// TIA Portal project "Program_PLC_LEGO" (V18)

(* hardware
DEVICE "S7-1200 station_1"  S7-1200 Station
   slot 0: "Rack_0"  S7-1200 Rack  Rack  V1.0
   slot 1: "PLC_1"  CPU 1214C DC/DC/DC  6ES7 214-1AG40-0XB0  V4.6
DEVICE "master"  GSD.Device.PN
   slot 0: "Rack"  Rack  V1.0
   slot 0: "bnixg35080b5r067"  BNI XG3-508-0B5-R067  BNI00L3  V1.3.2
      slot 0: "BNI XG3-508-0B5-R067"  BNI XG3-508-0B5-R067
      slot 1: "PN-IO"  PN-IO
         slot 1: "Port XF1"  Port XF1
         slot 2: "Port XF2"  Port XF2
   slot 1: "IO-Link I/O Ports_1"  IO-Link I/O Ports
      slot 0: "BALLUFF 8 Port IO-Link Master"  BALLUFF 8 Port IO-Link Master
   slot 1: "Digital Input"  Digital Input
   slot 2: "Digital Input_1"  Digital Input
   slot 3: "IOL_I/O_10/10_Byte + PQI_2"  IOL_I/O_10/10_Byte + PQI
   slot 4: "IOL_I/O_10/10_Byte + PQI_3"  IOL_I/O_10/10_Byte + PQI
   slot 5: "IOL_I/O_10/10_Byte + PQI_1"  IOL_I/O_10/10_Byte + PQI
   slot 6: "IOL_I/O_10/10_Byte + PQI"  IOL_I/O_10/10_Byte + PQI
   slot 7: "BNI IOL-302-S02-X026"  BNI IOL-302-S02-X026
   slot 8: "IOL_I/O_32/32_Byte + PQI"  IOL_I/O_32/32_Byte + PQI
*)

// ===== PLC "PLC_1"  CPU 1214C DC/DC/DC =====

VAR_GLOBAL   // PLC tag table "Default tag table"
   "Tag_1" AT %I68.0 : Bool;
   "Tag_2" AT %I68.1 : Bool;
   "RFID1" AT %I96.0 : Bool;   // rfid1
   "Tag_4" AT %M10.0 : Bool;
   "Tag_5" AT %ID98 : DWord;
   "Tag_6" AT %QB96 : Byte;
   "Tag_7" AT %M10.1 : Bool;
   "RFID2" AT %I107.0 : Bool;
   "RFID3" AT %I85.0 : Bool;
   "RFID4" AT %I74.0 : Bool;
   "Tag_8" AT %I68.2 : Bool;
   "Tag_9" AT %I68.3 : Bool;
   "Tag_10" AT %I3.0 : Bool;
   "Tag_11" AT %I4.0 : Bool;
END_VAR

TYPE "udtZlecenia"
   STRUCT
      Zlecenie : Struct
         ID : Int;   // Numer zlecenia
         Model : Int;   // Rodzaj modelu 2-8
         PartNo : Int;   // Nr sztuki
         "Time" : Struct   // Czasy na stanowiskach
            Stanowisko1 : Struct
               StartTime : DTL;   // Czas rozpoczecia
               EndTime : DTL;   // Czas zakonczenia
               TargetTime : Int;   // Zakladany czas
               ActualTime : Int;
               Abort : Bool;   // Czy anulowano produkcje na tym stanowisku
            END_STRUCT;
            Stanowisko2 : Struct
               StartTime : DTL;   // Czas rozpoczecia
               EndTime : DTL;   // Czas zakonczenia
               TargetTime : Int;   // Zakladany czas
               ActualTime : Int;
               Abort : Bool;   // Czy anulowano produkcje na tym stanowisku
            END_STRUCT;
            Stanowisko3 : Struct
               StartTime : DTL;   // Czas rozpoczecia
               EndTime : DTL;   // Czas zakonczenia
               TargetTime : Int;   // Zakladany czas
               ActualTime : Int;
               Abort : Bool;   // Czy anulowano produkcje na tym stanowisku
            END_STRUCT;
            StanowiskoQC : Struct
               StartTime : DTL;   // Czas rozpoczecia
               EndTime : DTL;   // Czas zakonczenia
               TargetTime : Int;   // Zakladany czas
               ActualTime : Int;
               Abort : Bool;   // Czy anulowano produkcje na tym stanowisku
            END_STRUCT;
         END_STRUCT;
         Alarm : Struct
            Stanowisko1 : Struct
               MissingPart : Bool;
               DamagedPart : Bool;
               PalletFault : Bool;
               WrongInstruction : Bool;
               SensorFault : Bool;
               Other : Bool;
            END_STRUCT;
            Stanowisko2 : Struct
               MissingPart : Bool;
               DamagedPart : Bool;
               PalletFault : Bool;
               WrongInstruction : Bool;
               SensorFault : Bool;
               Other : Bool;
            END_STRUCT;
            Stanowisko3 : Struct
               MissingPart : Bool;
               DamagedPart : Bool;
               PalletFault : Bool;
               WrongInstruction : Bool;
               SensorFault : Bool;
               Other : Bool;
            END_STRUCT;
            StanowieskoQC : Struct
               Camera : Bool;
               NOK : Bool;
               PalletFault : Bool;
               RFID : Bool;
               SensorFault : Bool;
               Other : Bool;
            END_STRUCT;
         END_STRUCT;
         ReturnQC : Bool;   // True - poprawny wyrób, False zły wyrób
         Priority : Int;   // 0 - Najniższy, 5 - Najwyższy
         Status : Array[0..3] of Bool;   // Status czy skonczono na danym stanowisku
         NOK : Struct
            NoBrick : Bool;
            WrongColour : Bool;
            Offset : Bool;
            Damage : Bool;
            WrongNumber : Bool;
            Other : Bool;
         END_STRUCT;
      END_STRUCT;
   END_STRUCT;
END_TYPE

TYPE "udtStanowiskoAssembly"
   STRUCT
      Config : Struct
         ID : Int;
         "Name" : String[20];
         HorlyRate : Real;
      END_STRUCT;
      Production : Struct
         State : Int;   // 0 - Gotowy. 1 - Montaż, 2 - Zakończono, 3 - Awaria
         OrderNo : Int;
         ProductNo : Int;
      END_STRUCT;
      "Time" : Struct
         TargetTime : Time;
         LastSec : UInt;
         RemainingSec : Int;
         RemainingStr : String[6];
         Blink : Bool;
      END_STRUCT;
      Commands : Struct
         Start : Struct
            Enable : Bool;
            State : Bool;
         END_STRUCT;
         FInish : Struct
            Enable : Bool;
            State : Bool;
         END_STRUCT;
         ReportFault : Struct
            Enable : Bool;
            State : Bool;
         END_STRUCT;
         AbortProcess : Struct
            Enable : Bool;
            State : Bool;
         END_STRUCT;
         FaultReason : Struct
            MissingPart : Bool;
            DamagedPart : Bool;
            PalletFault : Bool;
            WrongInstruction : Bool;
            SensorFault : Bool;
            Other : Bool;
         END_STRUCT;
      END_STRUCT;
      Sensors : Struct
         PalletPresent : Bool;
         RFID : Struct
            TagPresent : Bool;
            CmdRead : Bool;
            CmdWrite : Bool;
            Status : Bool;
            OrderNo : Int;
            ProductNo : Int;
         END_STRUCT;
      END_STRUCT;
      Stats : Struct
         DoneToday : Int;
         Efficiency : Int;
         ActudalPart : Int;
         Instruction : Int;
         Loaded : Bool;
      END_STRUCT;
      HMI : Struct
         Clear : Bool;   // Czyści licznik
         Container : Array[1..3] of Struct   // Tablica kontenerów
            value : Int;   // Ilość kontenerów 0 - 3
            Add : Struct   // Impuls na reczne dodanie
               Enable : Bool;
               Status : Bool;
            END_STRUCT;
            Subtract : Struct   // Impuls na reczne odejmowanie
               Enable : Bool;
               Status : Bool;
            END_STRUCT;
         END_STRUCT;
      END_STRUCT;
      MontazState : Int;
   END_STRUCT;
END_TYPE

TYPE "udtDbKomunikacja"
   STRUCT
      Trigger : Bool;
      NumerZlecenia : String[50];
      NumerOperacji : DInt;
      NumerPaletki : String[50];
      Stanowisko : String[50];
      Operator : String[50];
      CzasCykluMs : DInt;
      WynikQC : Bool;
      IloscWyprodukowanych : DInt;
      LiczbaWadliwych : DInt;
      KodPostoju : String[20];
   END_STRUCT;
END_TYPE

DATA_BLOCK "DB_Data"   // DB1
{ S7_Optimized_Access := 'FALSE' }
VERSION : 0.1
   VAR
      Stanowisko1 : "udtStanowiskoAssembly";
      Stanowisko2 : "udtStanowiskoAssembly";
      Stanowisko3 : "udtStanowiskoAssembly";
      StanowiskoQC : Struct
         Config : Struct
            ID : Int;
            "Name" : String[20];
            HorlyRate : Real;
         END_STRUCT;
         Production : Struct
            State : Int;
            OrderNo : Int;
            ProductNo : Int;
         END_STRUCT;
         "Time" : Struct
            TargetTime : Time;
            LastSec : UInt;
            RemainingSec : Int;
            RemainingStr : String[6];
            Blink : Bool;
         END_STRUCT;
         Commands : Struct
            Start : Struct
               Enable : Bool;
               State : Bool;
            END_STRUCT;
            OK : Struct
               Enable : Bool;
               State : Bool;
            END_STRUCT;
            NOK : Struct
               Enable : Bool;
               State : Bool;
               NoBrick : Bool;
               WrongColour : Bool;
               Offset : Bool;
               Damage : Bool;
               WrongNumber : Bool;
               Other : Bool;
            END_STRUCT;
            ReportFault : Struct
               Enable : Bool;
               State : Bool;
            END_STRUCT;
         END_STRUCT;
         Sensors : Struct
            PalletPresent : Bool;
            RFID : Struct
               TagPresent : Bool;
               CmdRead : Bool;
               CmdWrite : Bool;
               Status : Bool;
               OrderNo : Int;
               ProductNo : Int;
            END_STRUCT;
         END_STRUCT;
         Stats : Struct
            DoneToday : Int;
            Efficiency : Int;
            ActudalPart : Int;
            Instruction : Int;
            Loaded : Bool;
            PartsOK : Int;
            PartsNOK : Int;
            PartsPercent : Int;
         END_STRUCT;
         HMI : Struct
            Clear : Bool;
            CameraStatus : Int;
         END_STRUCT;
         QualityState : Int;
         FaultReason : Struct
            Camera : Bool;
            NOK : Bool;
            PalletFault : Bool;
            RFID : Bool;
            SensorFault : Bool;
            Other : Bool;
         END_STRUCT;
         CameraControl : Struct
            bInit : Bool;
            bGetResult : Bool;
            bResetError : Bool;
            wynikOK : Bool;
            bReq : Bool;
            bTrigger : Bool;
            bZrobInspekcje : Bool;
            krok : Int;
            wynikOV : Array[0..5] of Bool;
            CameraStatus : Bool;
         END_STRUCT;
      END_STRUCT;
      ZlecenieIndex : Array[0..3] of Int;
      DoneAllTime : Array[0..3] of Int;
   END_VAR
BEGIN
   Stanowisko1.Production.State := 0;
   Stanowisko1.Production.OrderNo := 0;   // Nr zlecenia
   // Stanowisko1.Config.ID : ID stanowiska
   // Stanowisko1.Config."Name" : Nazwa stanowiska
   // Stanowisko1.Config.HorlyRate : Stawka godzinowa
   // Stanowisko1.Production.ProductNo : Nr modelu
   // Stanowisko1."Time".TargetTime : Zakładany czas ukończenia wyrobu
   // Stanowisko1."Time".RemainingSec : pozostałe sekundy
   // Stanowisko1."Time".RemainingStr : sekundy w string
   // Stanowisko1.Commands : komendy
END_DATA_BLOCK

DATA_BLOCK "DB_PTL"   // DB2
{ S7_Optimized_Access := 'FALSE' }
VERSION : 0.1
   VAR
      PTL_state : Array[0..8] of Bool;
      Stanowisko : Array[0..2] of Struct
         Row1 : Int;   // 0 - brak, 3 - wszytskie kontenery
         Row2 : Int;   // 0 - brak, 3 - wszytskie kontenery
         Row3 : Int;   // 0 - brak, 3 - wszytskie kontenery
      END_STRUCT;
      ConnParams : TCON_IP_v4;
      InitDone : Bool;
      Wyzwalacz : Bool;
      mb_done : Bool;
      mb_busy : Bool;
      mb_error : Bool;
      mb_status : Word;
      PTL_Buttons : Array[1..9] of Word;
      PTL_State_Old : Array[0..8] of Bool;
   END_VAR
BEGIN
   // PTL_state[0] : Stanowisko 1.1
   // PTL_state[1] : Stanowisko 1.2
   // PTL_state[2] : Stanowisko 1.3
   // PTL_state[3] : Stanowisko 2.1
   // PTL_state[4] : Stanowisko 2.2
   // PTL_state[5] : Stanowisko 2.3
   // PTL_state[6] : Stanowisko 3.1
   // PTL_state[7] : Stanowisko 3.2
   // PTL_state[8] : Stanowisko 3.3
END_DATA_BLOCK

DATA_BLOCK "DB_Zlecenia"   // DB3
{ S7_Optimized_Access := 'FALSE' }
VERSION : 0.1
   VAR
      Zlecenie : Array[0..199] of "udtZlecenia";
      NastepneZlecenie : "udtZlecenia";
      PusteZlecenie : "udtZlecenia";   // Nie dopisywac wartosci!!!
      ResetZlecen : Bool;
   END_VAR
BEGIN
END_DATA_BLOCK

DATA_BLOCK "DB_WWW"   // DB5
{ S7_Optimized_Access := 'FALSE' }
VERSION : 0.1
   VAR
      Comm : "udtDbKomunikacja";
   END_VAR
BEGIN
END_DATA_BLOCK

DATA_BLOCK "BIS_V_CLM_COM_DB"   // DB6
{ S7_Optimized_Access := 'TRUE' }
AUTHOR : BICU
FAMILY : Ident
VERSION : 1.0
// stored: InstanceOfName BIS_V_CLM_COM
"BIS_V_CLM_COM"
BEGIN
END_DATA_BLOCK

DATA_BLOCK "RFID_test"   // DB7
{ S7_Optimized_Access := 'TRUE' }
VERSION : 0.1
   VAR
      Bufor_Odczyt : Array[0..10] of Byte;
      Bufor_Zapis : Array[0..10] of Byte;
      Bufor_Odczyt2 : Array[0..10] of Byte;
      Bufor_Odczyt3 : Array[0..10] of Byte;
      Bufor_Odczyt4 : Array[0..10] of Byte;
   END_VAR
BEGIN
END_DATA_BLOCK

DATA_BLOCK "BIS_V_CLM_COM_DB_1"   // DB8
{ S7_Optimized_Access := 'TRUE' }
AUTHOR : BICU
FAMILY : Ident
VERSION : 1.0
// stored: InstanceOfName BIS_V_CLM_COM
"BIS_V_CLM_COM"
BEGIN
END_DATA_BLOCK

DATA_BLOCK "BIS_V_CLM_COM_DB_2"   // DB9
{ S7_Optimized_Access := 'TRUE' }
AUTHOR : BICU
FAMILY : Ident
VERSION : 1.0
// stored: InstanceOfName BIS_V_CLM_COM
"BIS_V_CLM_COM"
BEGIN
END_DATA_BLOCK

DATA_BLOCK "DB_Cam_Input"   // DB10
{ S7_Optimized_Access := 'FALSE' }
VERSION : 0.1
   VAR
      Input : Array[0..127] of Byte;
   END_VAR
BEGIN
END_DATA_BLOCK

DATA_BLOCK "DB_Cam_Output"   // DB11
{ S7_Optimized_Access := 'FALSE' }
VERSION : 0.1
   VAR
      Output : Array[0..127] of Byte;
   END_VAR
BEGIN
END_DATA_BLOCK

DATA_BLOCK "BVS_Sensor_DB"   // DB12
{ S7_Optimized_Access := 'TRUE' }
AUTHOR : PD-ILS
FAMILY : Balluff
VERSION : 1.1
// stored: InstanceOfName BVS_Sensor
"BVS_Sensor"
BEGIN
END_DATA_BLOCK

DATA_BLOCK "BIS_V_CLM_COM_DB_3"   // DB13
{ S7_Optimized_Access := 'TRUE' }
AUTHOR : BICU
FAMILY : Ident
VERSION : 1.0
// stored: InstanceOfName BIS_V_CLM_COM
"BIS_V_CLM_COM"
BEGIN
END_DATA_BLOCK

FUNCTION_BLOCK "RaportowanieDB"   // FB1, SCL
{ S7_Optimized_Access := 'TRUE' }
VERSION : 0.1
   VAR_TEMP
      temp_CzasObecny : Int;
      temp_DTL : Int;
      temp_RoznicaCzasu : Time;
   END_VAR
BEGIN
   // Uruchamiaj tylko, gdy C# potwierdził odebranie poprzednich danych (Trigger = 0)
   IF NOT "DB_WWW".Comm.Trigger THEN

       // ============================================
       // STANOWISKO 1 (Montażowe)
       // ============================================
       IF "DB_Data".Stanowisko1.Commands.FInish.State THEN

          // #temp_CzasObecny := RD_SYS_T(OUT => #temp_DTL);
          // #temp_RoznicaCzasu := T_DIFF(IN1 := #temp_DTL, IN2 := "DB_Data".Stanowisko1."Time".StartStamp);
           "DB_WWW".Comm.CzasCykluMs := TIME_TO_DINT(#temp_RoznicaCzasu);

           "DB_WWW".Comm.NumerZlecenia := 'ZL-2137'; // do podmiany na aktualne zlecenie
           "DB_WWW".Comm.Stanowisko := 'Assembly 1';
           "DB_WWW".Comm.Operator := 'Operator 1';
           "DB_WWW".Comm.IloscWyprodukowanych := 1;

           IF "DB_Data".Stanowisko1.Commands.FaultReason.DamagedPart THEN
               "DB_WWW".Comm.KodPostoju := 'DAMAGED_PART';
               "DB_WWW".Comm.WynikQC := FALSE;
               "DB_WWW".Comm.LiczbaWadliwych := 1;
           ELSIF "DB_Data".Stanowisko1.Commands.FaultReason.MissingPart THEN
               "DB_WWW".Comm.KodPostoju := 'MISSING_PART';
               "DB_WWW".Comm.WynikQC := FALSE;
               "DB_WWW".Comm.LiczbaWadliwych := 1;
           ELSE
               "DB_WWW".Comm.KodPostoju := '';
               "DB_WWW".Comm.WynikQC := TRUE;
               "DB_WWW".Comm.LiczbaWadliwych := 0;
           END_IF;

           "DB_WWW".Comm.Trigger := TRUE;
           "DB_Data".Stanowisko1.Production.State := 2;
           "DB_Data".Stanowisko1.Commands.FInish.State := FALSE;

           // ============================================
           // STANOWISKO 2 (Montażowe)
           // ============================================
         //  ELSIF "DB_Data".Stanowisko2.Commands.FInish.State THEN

           //    #temp_CzasObecny := RD_SYS_T(OUT => #temp_DTL);
           //    #temp_RoznicaCzasu := T_DIFF(IN1 := #temp_DTL, IN2 := "DB_Data".Stanowisko2."Time".StartStamp);
            //   "DB_WWW".Comm.CzasCykluMs := TIME_TO_DINT(#temp_RoznicaCzasu);

            //   "DB_WWW".Comm.NumerZlecenia := 'ZL-2137';
            //   "DB_WWW".Comm.Stanowisko := 'Assembly 2';
            //   "DB_WWW".Comm.Operator := 'Operator 2';
            //   "DB_WWW".Comm.IloscWyprodukowanych := 1;

            //   IF "DB_Data".Stanowisko2.Commands.FaultReason.DamagedPart THEN
            //       "DB_WWW".Comm.KodPostoju := 'DAMAGED_PART';
            //       "DB_WWW".Comm.WynikQC := FALSE;
             //      "DB_WWW".Comm.LiczbaWadliwych := 1;
            //   ELSIF "DB_Data".Stanowisko2.Commands.FaultReason.MissingPart THEN
           //        "DB_WWW".Comm.KodPostoju := 'MISSING_PART';
           //        "DB_WWW".Comm.WynikQC := FALSE;
           //        "DB_WWW".Comm.LiczbaWadliwych := 1;
           //    ELSE
           //        "DB_WWW".Comm.KodPostoju := '';
           //        "DB_WWW".Comm.WynikQC := TRUE;
           //        "DB_WWW".Comm.LiczbaWadliwych := 0;
            //   END_IF;

            //   "DB_WWW".Comm.Trigger := TRUE;
            //   "DB_Data".Stanowisko2.Production.State := 2;
            //   "DB_Data".Stanowisko2.Commands.FInish.State := FALSE;

               // ============================================
               // STANOWISKO 3 (Montażowe)
               // ============================================
         //  ELSIF "DB_Data".Stanowisko3.Commands.FInish.State THEN

            //   #temp_CzasObecny := RD_SYS_T(OUT => #temp_DTL);
            //   #temp_RoznicaCzasu := T_DIFF(IN1 := #temp_DTL, IN2 := "DB_Data".Stanowisko3."Time".StartStamp);
            //   "DB_WWW".Comm.CzasCykluMs := TIME_TO_DINT(#temp_RoznicaCzasu);

            //   "DB_WWW".Comm.NumerZlecenia := 'ZL-2137';
           //    "DB_WWW".Comm.Stanowisko := 'Assembly 3';
            //   "DB_WWW".Comm.Operator := 'Operator 3';
            //   "DB_WWW".Comm.IloscWyprodukowanych := 1;

           //    IF "DB_Data".Stanowisko3.Commands.FaultReason.DamagedPart THEN
           //        "DB_WWW".Comm.KodPostoju := 'DAMAGED_PART';
            //       "DB_WWW".Comm.WynikQC := FALSE;
             //      "DB_WWW".Comm.LiczbaWadliwych := 1;
            //   ELSIF "DB_Data".Stanowisko3.Commands.FaultReason.MissingPart THEN
            //       "DB_WWW".Comm.KodPostoju := 'MISSING_PART';
           //        "DB_WWW".Comm.WynikQC := FALSE;
           ///        "DB_WWW".Comm.LiczbaWadliwych := 1;
           //    ELSE
           //        "DB_WWW".Comm.KodPostoju := '';
           //        "DB_WWW".Comm.WynikQC := TRUE;
           //        "DB_WWW".Comm.LiczbaWadliwych := 0;
           //    END_IF;

           //    "DB_WWW".Comm.Trigger := TRUE;
            //   "DB_Data".Stanowisko3.Production.State := 2;
             //  "DB_Data".Stanowisko3.Commands.FInish.State := FALSE;

               // ============================================
               // STANOWISKO 4 (QC - Kontrola Jakości)
               // ============================================
         //  ELSIF "DB_Data".StanowiskoQC.Commands.FInish.State THEN

             //  #temp_CzasObecny := RD_SYS_T(OUT => #temp_DTL);
             //  #temp_RoznicaCzasu := T_DIFF(IN1 := #temp_DTL, IN2 := "DB_Data".StanowiskoQC."Time".StartStamp);
            //   "DB_WWW".Comm.CzasCykluMs := TIME_TO_DINT(#temp_RoznicaCzasu);

             //  "DB_WWW".Comm.NumerZlecenia := 'ZL-2137';
             //  "DB_WWW".Comm.Stanowisko := 'QC Station';
             //  "DB_WWW".Comm.Operator := 'Operator QC';

               // Zależnie od tego, jak raportujecie odrzuty na QC
              // IF "DB_Data".StanowiskoQC.Commands.FaultReason.DamagedPart THEN
              //     "DB_WWW".Comm.IloscWyprodukowanych := 0;
              //     "DB_WWW".Comm.KodPostoju := 'DAMAGED_PART';
              //     "DB_WWW".Comm.WynikQC := FALSE;
              //     "DB_WWW".Comm.LiczbaWadliwych := 1;
              // ELSE
              //     "DB_WWW".Comm.IloscWyprodukowanych := 1;
               //    "DB_WWW".Comm.KodPostoju := '';
               //    "DB_WWW".Comm.WynikQC := TRUE;
             //      "DB_WWW".Comm.LiczbaWadliwych := 0;
             //  END_IF;

             //  "DB_WWW".Comm.Trigger := TRUE;
               //"DB_Data".StanowiskoQC.Production.State := 2;
               //"DB_Data".StanowiskoQC.Commands.FInish.State := FALSE;

       END_IF;

   END_IF;
END_FUNCTION_BLOCK

FUNCTION_BLOCK "BIS_V_CLM_COM"   // FB33, SCL
TITLE = BIS V (VM, C, VL), BIS C, BIS M; BIS L Function Block
{ S7_Optimized_Access := 'TRUE' }
AUTHOR : BICU
FAMILY : Ident
VERSION : 1.0
   VAR_INPUT
      Init : Bool := FALSE;   // Internal reset and initailisation of FB
      Start : Bool := FALSE;   // Start command
      ProcReset : Bool := FALSE;   // Reset of BIS and FB
      HeadOff : Bool := FALSE;   // Head deactivation
      Dynamic : Bool := FALSE;   // Dynamic read / write function
      HW_LADDR : Hw_SubModule;   // HW_Address for cyclic com, BIS Module
      HW_LADDR_Q : Hw_SubModule;   // HW_Address for cyclic com, BIS Output Module
      Command : Int := 0;   // 1=Read; 2=Write;
      DB_Send : DB_ANY;
      Offset_DBSend : DInt := 0;   // Offset write data
      DB_Receive : DB_ANY;
      Offset_DBReceive : DInt := 0;   // Offset read data
      TAG_StartAddr : DInt := DINT#0;   // Start address from data carrier or parameter number
      TAG_NumbOfByte : DInt := DINT#0;   // Data lenght to be written or read or parameter Bytes
      WatchdogTime : Time := T#3S;   // Watchdog of commado
      CopTargetAddr : DInt;   // Traget Address for Copy Command
      CopRW_HeadNo : Int;   // Head number for Copy Command
      ProcType : Char := 'v';   // Processor Type V= BIS-V only | C, L, M = BIS * | I = BIS-M4** IO-Link
      OptIoLen : UInt := 10;   // Optional IO Length for IO-Link and C, L, M
      OptIoBuffOffs : UInt;   // IO Buffer offset for BIS C, L, M, 2nd R/W head
   END_VAR
   VAR_OUTPUT
      Ready : Bool := FALSE;   // Command ready
      Error : Bool := FALSE;   // Command error
      ErrorCode : Word := 0;   // Error code
      MT : Bool := FALSE;   // Antenna selection is on
      DatCarrPresent : Bool := FALSE;   // Data Carrier present
   END_VAR
   VAR_IN_OUT
      DB_SendOpt : Variant;   // Data block write data
      DB_ReceiveOpt : Variant;   // Data block for read data
   END_VAR
   VAR
      PointerByte : DInt := 0;   // Pointer DB RW-Address
      LengthByte : DInt := 0;   // Number of bytes read/write per cycle
      BytePerPage : DInt := 0;   // Databytes lenght in IO buffer
      TotalByte : DInt := 0;   // Remaining all Byte data to be read/write
      HW_Init : Bool;   // Hardware adresses initialized
      ReadActive : Bool := FALSE;   // Read command active
      WriteActive : Bool := FALSE;   // Write command active
      ResetActive : Bool := FALSE;   // FB and Processor reset active
      ToggleOld : Bool := FALSE;   // Last state toggle-bit
      FirstCycle : Bool := FALSE;   // First read/write cycle
      IMP_Start : Bool := FALSE;   // Pulse bit Start
      ShortCom : Bool := FALSE;   // Command with 1 Byte data-length active
      RdLengIn : Bool;   // Read length info from input
      WriteCom : Bool := FALSE;   // Write command without data active
      CopyTag : Bool := FALSE;   // Copy Tag commando
      HeadOffActive : Bool := FALSE;   // AntSelBusy
      WaitOnAE : Bool;   // Read on AE Bit
      IOLink_Proc : Bool;   // BIS IO-Link processor M-4**-0**-001
      IOLink_Proc401 : Bool;   // BIS IO-Link processor M-4**-0**-401
      CLM_Proc : Bool;   // BIS classic C, L, M processor unit
      C_Cttp : Bool;   // BIS C Tag Type. False 32 Byte. True 64 Byte
      bHd_CP_CodePresent : Bool;   // Bit header In: Tag Present
      bHd_AA_JobStart : Bool;   // Bit header In: Job Start
      bHd_AE_JobEnd : Bool;   // Bit header In: Job End
      bHd_AF_JobError : Bool;   // Bit header In: Job Error
      bHd_MT_MultTag : Bool;   // Bit header In: Multiple Tags
      bHd_TO_ToggleOut : Bool;   // Bit header In: Toggle Bit Out
      bHd_HF_HeadFault : Bool;   // Bit header In: Head Fault
      bHd_BB_Ready : Bool;   // Bit header In: Ready for Operation
      bHd_AV_JobStart : Bool;   // Bit header Out: Job Start
      bHd_GR_Default : Bool;   // Bit header Out: Default State
      bHd_HD_HeadSel : Bool;   // Bit header Out: Head Selection BIS U
      bHd_KA_HeadOff : Bool;   // Bit header Out: Head shutoff
      bHd_TI_ToggleIn : Bool;   // Bit header Out: Togle Bit In
      bHd_Cttp_TagType : Bool;
      ProcRes_Int : Bool;   // Processor reset internal
      ErrorInt : Bool;   // Error bit internal
      ArrayInput : Array[0..#InBuSi] of Byte;   // BIS out to PLC in
      ArrayOutput : Array[0..#OutBuSi] of Byte;   // PLC out to BIS in
      R_TRIG_Start : R_TRIG;
      R_TRIG_Reset : R_TRIG;
      R_TRIG_KA : R_TRIG;
      F_TRIG_KA : F_TRIG;
      WD_Timer : TON_TIME;
      HF_Timer : TON_TIME;
      PIaddr : UDInt;   // Input address
      PIcount : UInt;   // Input length
      PQaddr : UDInt;   // Output address
      PQcount : UInt;   // Output address
      RetVal_ModulDiag : Int;   // Return value modul diagnosis
      RetVal_RD_Addr : Int;   // Return value read address
      RetVal_RD_DP : Int;   // Return value read input data
      RetVal_WR_DP : Int;   // Return value write output data
      RetVal_Get_ErrID : Word;   // Return value get error ID
      RetValVarMove : Int;
      CNT_Diag : UInt;   // CNT_Modul Diag
      Diag_Out : DWord;   // Modul Diag
      BIS_STA : Struct   // BIS Statusword
         CP_DaCarrPres : Bool := FALSE;   // Data Carrier present
         reserved_1 : Bool := FALSE;
         reserved_2 : Bool := FALSE;
         reserved_3 : Bool := FALSE;
         ChainedCom : Bool := FALSE;
         reserved_5 : Bool := FALSE;
         Error : Bool := FALSE;   // Error output set
         Ready : Bool := FALSE;   // FB Ready
         ResetAct : Bool := FALSE;   // Reset running
         Command_start : Bool := FALSE;   // FB Start is set
         reserved_6 : Bool := FALSE;
         InitAct : Bool := TRUE;   // Init running
         HF_Bit : Bool := FALSE;   // Head fault
         Busy : Bool := FALSE;   // Comando busy
         Reserved_7 : Bool := FALSE;
         Reserved_8 : Bool := FALSE;
         Com : Int := 0;   // 81=Read;82=Write; 42=Read EPC; 44=Read TID
         TStartAddr : DInt := DINT#0;   // Start address from data carrier or parameter number for diagnosis
         TNumbOfByte : DInt := DINT#0;   // data lenght to be written or read or parameter Bytes for diagnosis
      END_STRUCT;
      testdword : DWord;
   END_VAR
   VAR_TEMP
      tError : Word;   // temp Error number buffer
      tBTimeoutIN : Bool;   // temp Timeout in
      tBTimeoutQ : Bool;   // temp Timeout output
      tLoop : DInt;   // temp Loop counter
      tempDB : DB_ANY;
      tUdint : UDInt;
      tLCnt : UDInt;
      tVariant : Variant;
      tErrorConvVar : Int;
      tempTest : DB_ANY;
      tWordTest : Word;
      tempDBErr : Int;
   END_VAR
   VAR CONSTANT
      InBuSi : Int := 254;   // maximum size inputbuffer
      OutBuSi : Int := 254;   // maximum size outputbuffer
   END_VAR
BEGIN
   //=============================================================================
   //Balluff GmbH
   //(c)Copyright (2019) All Rights Reserved
   //-----------------------------------------------------------------------------
   //Library: BIS_V
   //Tested with: CPU 1214C V4.1
   //Engineering: TIA Portal V13 SP1 
   //Restrictions: -
   //Requirements: PLC (S7-1200 / S7-1500)
   //Functionality: RFID commandos for BIS V, BIS C, BIS M, BIS L processor units
   //-----------------------------------------------------------------------------
   //Change log table:
   //Version  Date       Expert in charge  Changes applied
   //
   //00.01.00 18.03.2019 Balluff GmbH PD   First created with TIA V13 SP1 with mem opt
   //=============================================================================
   //
   (*
   Disclaimer of Liability
   **********************
   The demo function block is free of charge and is a universal application 
   example.
   This demo function block shall help program and configure PLC applications and 
   shall provide possible solutions.
   The user is not entitled to claim for warranty, error correction and updates. 
   In 
   particular there is excluded any claims against Balluff GmbH for damages that 
   might result from the use of this demo program. Excluded from this limitation 
   of 
   liability shall be (a) those damages that are based on injury to life, limb or 
   health, (b) a liability according to the Produkthaftungsgesetz (German Product 
   Liability Law) and (c) cases of willful intent.
   Please check if the function block is intended for your application before 
   adapting it in plants and machineries.
   By using the S7 sample, made available free of charge you accept the limitation 
   of 
   warranty and liability!

   Haftungsausschluss:
   *********************
   Der hier kostenlos verfügbare DEMO-Baustein ist ein allgemeingültiges 
   Anwendungsbeispiel. Dieser DEMO-Baustein soll bei der Programmierung und 
   Projektierung von SPS-Anwendungen unterstützen und Lösungsansätze aufzeigen. 
   Ein Anspruch auf Gewährleistung, Fehlerbeseitigung und Update besteht für den 
   Anwender nicht. Die BALLUFF GmbH schließt insbesondere jegliche Haftung für 
   Schäden, die durch den Einsatz dieses DEMO-Bausteins entstehen, ausdrücklich 
   aus! Diese Haftungsbeschränkung gilt nicht bei Verletzungen des Lebens, des 
   Körpers oder der Gesundheit, bei der Haftung nach dem Produkthaftungsgesetz und 
   bei vorsätzlichen Pflichtverletzungen. 
   Prüfen Sie vor dem Einsatz in Anlagen und Maschinen, ob der hier 
   bereitgestellte 
   DEMO Baustein für Ihre Anwendung nutzbar ist!
   Mit dem Einsatz des hier kostenlos vorgelegten S7-Beispiel erkennen Sie die 
   Gewährleistungs- und Haftungsbegrenzung an!

       *)

   //-----------------------------------------------------------------------------
   //Select Processor unit
   //-----------------------------------------------------------------------------


   // Default select BIS V
   IF (#ProcType = 'V') OR
     (#ProcType = 'v') THEN
     #WaitOnAE := FALSE;
     #IOLink_Proc := FALSE;
     #CLM_Proc := FALSE;
     #IOLink_Proc401 := FALSE;

     // Select BIS C, L, M processor    
   ELSIF (#ProcType = 'M') OR // M upper case
     (#ProcType = 'm') OR // m lower case
     (#ProcType = 'C') OR // C upper case
     (#ProcType = 'c') OR // c lower case
     (#ProcType = 'L') OR // L upper case
     (#ProcType = 'l') THEN // l lower case
     #WaitOnAE := TRUE;
     #IOLink_Proc := FALSE;
     #CLM_Proc := TRUE;
     #IOLink_Proc401 := FALSE;

     // Select BIS IO-Link compact processor unit    
   ELSIF (#ProcType = 'I') OR  // I upper case
     (#ProcType = 'i') THEN  // i lower case
     #WaitOnAE := TRUE;
     #IOLink_Proc := TRUE;
     #CLM_Proc := FALSE;
     #IOLink_Proc401 := FALSE;

     // Select BIS IO-Link compact processor unit   BIS M-4xx-xxx-401 
   ELSIF (#ProcType = 'K') OR  // I upper case
     (#ProcType = 'k') THEN  // i lower case
     #WaitOnAE := TRUE;
     #IOLink_Proc := TRUE;
     #CLM_Proc := FALSE;
     #IOLink_Proc401 := TRUE;

     // Siemens Master BIS M-4xx-xxx-001        
   ELSIF (#ProcType = 'X') OR  // I upper case
     (#ProcType = 'x') THEN  // i lower case
     #WaitOnAE := TRUE;
     #IOLink_Proc := TRUE;
     #CLM_Proc := TRUE;
     #IOLink_Proc401 := FALSE;

     // Siemens Master BIS M-4xx-xxx-401     
   ELSIF (#ProcType = 'Y') OR  // I upper case
     (#ProcType = 'y') THEN  // i lower case
     #WaitOnAE := TRUE;
     #IOLink_Proc := TRUE;
     #CLM_Proc := TRUE;
     #IOLink_Proc401 := TRUE;

   END_IF;

   // Select tag type for C System
   IF ((#ProcType = 'C') OR // C upper case
     (#ProcType = 'c')) AND // c lower case
     #C_Cttp THEN
     #bHd_Cttp_TagType := TRUE;
   ELSE
     #bHd_Cttp_TagType := FALSE;
   END_IF;

   //-------------------------------------------------
   // HMI Out
   //-------------------------------------------------
   #BIS_STA.CP_DaCarrPres := #bHd_CP_CodePresent;
   #BIS_STA.HF_Bit := #bHd_HF_HeadFault;
   #BIS_STA.InitAct := #Init;
   #BIS_STA.Error := #ErrorInt;

   #BIS_STA.ResetAct := #ResetActive;
   //-----------------------------------------------------------------------------
   //FB Init, reset static variables
   //-----------------------------------------------------------------------------
   IF #Init THEN
     #PointerByte := 0;
     #LengthByte := 0;
     #BytePerPage := 0;
     #TotalByte := 0;
     #ReadActive := FALSE;
     #WriteActive := FALSE;
     #ResetActive := FALSE;
     #ToggleOld := FALSE;
     #FirstCycle := FALSE;
     #ShortCom := FALSE;
     #WriteCom := FALSE;
     #Ready := TRUE;
     #Error := FALSE;
     #ErrorCode := 0;
     #HW_Init := FALSE;
     #HeadOffActive := FALSE;
     #ProcRes_Int := TRUE;
     #R_TRIG_Reset.Stat_Bit := FALSE;
   END_IF;

   //-----------------------------------------------------------------------------
   // read modul states
   //-----------------------------------------------------------------------------
   #RetVal_ModulDiag := GET_DIAG(MODE := 0, LADDR := #HW_LADDR, CNT_DIAG => #CNT_Diag, DIAG := #Diag_Out);

   //-----------------------------------------------------------------------------
   // reading PI/PQ addr and data length
   //-----------------------------------------------------------------------------
   IF NOT #HW_Init THEN
     #RetVal_RD_Addr := RD_ADDR(LADDR := #HW_LADDR, PIADDR => #PIaddr, PICount => #PIcount,
                                PQADDR => #PQaddr, PQCount => #PQcount);
     IF #IOLink_Proc THEN
       #PIcount := #OptIoLen;
       #PQcount := #OptIoLen;
     END_IF;

     IF #CLM_Proc THEN
       IF NOT #IOLink_Proc THEN
         #RetVal_RD_Addr := RD_ADDR(LADDR := #HW_LADDR_Q, PIADDR => #tUdint, PICount => #tUdint,
                                    PQADDR => #PQaddr, PQCount => #PQcount);
       END_IF;

       IF #OptIoBuffOffs = 0 THEN //1st Buffer selected
         #PQcount := #OptIoLen; // overwrite length
         #PIcount := #OptIoLen;
       ELSIF #OptIoBuffOffs <> 0 THEN //2nd Buffer selected
         #PQaddr := #PQaddr + #OptIoBuffOffs; // overwrite Address 
         #PQcount := #OptIoLen; // overwrite Address 
         #PIaddr := #PIaddr + #OptIoBuffOffs;
         #PIcount := #OptIoLen;
       END_IF;
     END_IF;

     #HW_Init := TRUE;
   END_IF;

   //-----------------------------------------------------------------------------
   // cyclic read cam input if HW init done
   //----------------------------------------------------------------------------- 
   IF #HW_Init THEN
     IF #CLM_Proc THEN
       #tLCnt := 0;
       #RetVal_RD_DP := 0;
       #RetVal_WR_DP := 0;
       FOR #tLoop := UDINT_TO_DINT(#PIaddr) TO UDINT_TO_DINT(#PIaddr + #PIcount) DO
         #ArrayInput[#tLCnt] := PEEK(area := 16#81, dbNumber := 0, byteOffset := #tLoop);
         #tLCnt := #tLCnt + 1;
       END_FOR;

     ELSE
       #RetVal_RD_DP := DPRD_DAT(LADDR := #HW_LADDR, RECORD => #ArrayInput);
     END_IF;
   END_IF;
   //-----------------------------------------------------------------------------
   // Comapre bitheader
   //-----------------------------------------------------------------------------
   IF #ArrayInput[0] <> #ArrayInput[#PIcount - 1] THEN
     RETURN;
   END_IF;

   //-----------------------------------------------------------------------------
   // Move input bytes to static bits
   //-----------------------------------------------------------------------------
   #bHd_CP_CodePresent := #ArrayInput[0].%X0;
   #bHd_AA_JobStart := #ArrayInput[0].%X1;
   #bHd_AE_JobEnd := #ArrayInput[0].%X2;
   #bHd_AF_JobError := #ArrayInput[0].%X3;
   #bHd_MT_MultTag := #ArrayInput[0].%X4;
   #bHd_TO_ToggleOut := #ArrayInput[0].%X5;
   #bHd_HF_HeadFault := #ArrayInput[0].%X6;
   #bHd_BB_Ready := #ArrayInput[0].%X7;

   //-------------------------------------------------
   // KA HeadOff
   //-------------------------------------------------
   #R_TRIG_KA(CLK := #HeadOff);
   #F_TRIG_KA(CLK := #HeadOff);
   IF #R_TRIG_KA.Q THEN    // Deactivate head
     #bHd_KA_HeadOff := TRUE;
     #Ready := FALSE;
     #DatCarrPresent := FALSE;
     #HeadOffActive := TRUE;
     GOTO DataOut;
   END_IF;

   IF #F_TRIG_KA.Q THEN    // Activate head
     #bHd_KA_HeadOff := FALSE;
     #Ready := FALSE;
     #HeadOffActive := FALSE;
     GOTO DataOut;
   END_IF;

   //-------------------------------------------------
   // FB Reset
   //-------------------------------------------------
   #R_TRIG_Reset(CLK := #ProcReset OR #ProcRes_Int);

   IF #R_TRIG_Reset.Q THEN
     #ResetActive := TRUE;
     #PointerByte := 0;
     #LengthByte := 0;
     #BytePerPage := 0;
     #TotalByte := 0;
     #ReadActive := FALSE;
     #WriteActive := FALSE;
     #ToggleOld := FALSE;
     #FirstCycle := FALSE;
     #ShortCom := FALSE;
     #WriteCom := FALSE;
     #CopyTag := FALSE;
     #Ready := FALSE;
     #bHd_GR_Default := TRUE;
     IF NOT #ProcRes_Int THEN
       #Error := FALSE;
       #ErrorCode := 0;
     END_IF;
     #ProcRes_Int := FALSE;
     #HeadOffActive := FALSE;
     GOTO DataOut;

   END_IF;

   IF #ResetActive AND NOT #bHd_BB_Ready THEN
     #bHd_GR_Default := false;
     #ResetActive := false;
     GOTO AV_Reset;
   END_IF;
   //-----------------------------------------------------------------------------
   // MT Multiple Tags; CT Present
   //-----------------------------------------------------------------------------
   #MT := #bHd_MT_MultTag;

   #DatCarrPresent := #bHd_CP_CodePresent;

   //-----------------------------------------------------------------------------
   // Command Start
   #R_TRIG_Start(CLK := #Start,
                 Q => #IMP_Start);
   //-----------------------------------------------------------------------------

   //-----------------------------------------------------------------------------
   // Check HW/Profinet Error when start is set
   //-----------------------------------------------------------------------------
   IF #IMP_Start THEN
     IF #RetVal_RD_Addr <> 0 THEN
       #tError := w#16#50; //Error read address
       GOTO Error;
     END_IF;

     IF #RetVal_RD_DP <> 0 THEN
       #tError := w#16#51; //Error read input data
       GOTO Error;
     END_IF;

     IF #RetVal_WR_DP <> 0 THEN
       #tError := w#16#52; //Error read output data
       GOTO Error;
     END_IF;

   END_IF;

   IF #bHd_AF_JobError AND NOT #ProcReset THEN // Check error
     #tError := #ArrayInput[1];
     GOTO Error;
   END_IF;

   #HF_Timer(IN := #bHd_HF_HeadFault AND (NOT #HeadOff OR (NOT #IOLink_Proc AND NOT #CLM_Proc)),
             PT := t#500ms);

   IF #HF_Timer.Q//Head fault timeout
     AND NOT #ProcReset
     AND (NOT #IOLink_Proc
     OR #IOLink_Proc
     AND NOT #HeadOff)
   THEN // Check head fault
     #tError := 16#09;
     GOTO Error;
   END_IF;

   IF #IMP_Start AND
     (#TAG_NumbOfByte > 65534) AND NOT
     (#Command = 16#B2) THEN
     #tError := w#16#84;
     GOTO Error;
   END_IF;

   //-----------------------------------------------------------------------------
   // FB ready output 
   //-----------------------------------------------------------------------------
   #Ready :=
   NOT #ReadActive AND
   NOT #WriteActive AND
   NOT #ResetActive AND
   NOT #ShortCom AND
   NOT #CopyTag AND
   NOT #WriteCom AND
   NOT #bHd_AA_JobStart AND
   NOT #bHd_AE_JobEnd AND
   NOT #bHd_AF_JobError AND
   NOT #HeadOffActive AND
   #bHd_BB_Ready;

   //-----------------------------------------------------------------------------
   // BIS status for HMI
   //-----------------------------------------------------------------------------
   #BIS_STA.Ready := #Ready;
   #BIS_STA.Command_start := #Start;
   #BIS_STA.Com := #Command;
   #BIS_STA.TStartAddr := #TAG_StartAddr;
   #BIS_STA.TNumbOfByte := #TAG_NumbOfByte;

   IF #BIS_STA.Ready THEN
     #BIS_STA.ResetAct := FALSE;
     #BIS_STA.Busy := FALSE;
   END_IF;
   //-----------------------------------------------------------------------------
   // Generate error timeout
   //-----------------------------------------------------------------------------
   #tBTimeoutIN := (NOT #Ready AND NOT #Dynamic
   AND NOT #ResetActive
   AND NOT #HeadOffActive
   AND NOT #ProcRes_Int);

   #WD_Timer(IN := #tBTimeoutIN,
             PT := #WatchdogTime,
             Q => #tBTimeoutQ);

   IF #tBTimeoutQ THEN
     #tError := w#16#80;
     #ProcRes_Int := #bHd_AA_JobStart;
     GOTO Error;
   END_IF;

   //=============================================================================
   //
   // Reader commandos
   //
   //=============================================================================

   //-----------------------------------------------------------------------------
   // Goto FB end if no job active
   //-----------------------------------------------------------------------------

   IF (NOT #ReadActive AND
     NOT #WriteActive AND
     NOT #ShortCom AND
     NOT #WriteCom AND
     NOT #CopyTag AND
     (NOT #IMP_Start OR
     NOT #Ready OR
     #bHd_AA_JobStart)) OR
     #HeadOffActive THEN
     RETURN;
   END_IF;

   IF #ReadActive THEN  // Check Get or Set
     GOTO Read;
   ELSIF #WriteActive THEN
     GOTO Write;
   ELSIF #WriteCom OR #CopyTag THEN
     GOTO WriteCom;
   END_IF;

   //-----------------------------------------------------------------------------
   // Initialize Command output
   //-----------------------------------------------------------------------------
   #ArrayOutput[3] := 0;
   #ArrayOutput[4] := 0;
   #ArrayOutput[5] := 0;
   #ArrayOutput[6] := 0;
   #ArrayOutput[7] := 0;
   #ArrayOutput[8] := 0;

   CASE #Command OF

     16#1: // Read user data       
       #ArrayOutput[1] := 16#1;
       #PointerByte := #Offset_DBReceive;
       #ReadActive := TRUE;
     16#2: // Write user data       
       #ArrayOutput[1] := 16#2;
       #PointerByte := #Offset_DBSend;
       #WriteActive := TRUE;
     16#7: // // Store Start address for Auto read
       #ArrayOutput[1] := 16#7;
       #WriteActive := TRUE;
       #WriteCom := TRUE;
     16#9: // Read Typ and Serial  
       #ArrayOutput[1] := 16#9;
       #PointerByte := #Offset_DBReceive;
       #RdLengIn := TRUE;
       #ReadActive := TRUE;
     16#11: // Copy data between data carriers
       #ArrayOutput[1] := 16#11;
       #PointerByte := #Offset_DBReceive;
       #WriteCom := TRUE;
       #TotalByte := 0;
     16#12: // Initialize CRC16       
       #ArrayOutput[1] := 16#12;
       #PointerByte := #Offset_DBSend;
       #WriteActive := TRUE;
     16#13: // Read DSFID
       #ArrayOutput[1] := 16#13;
       #PointerByte := #Offset_DBReceive;
       #TotalByte := 1;
       #ReadActive := TRUE;
     16#14: // Write DSFID
       #ArrayOutput[1] := 16#14;
       #PointerByte := #Offset_DBReceive;
       #TotalByte := 1;
       #WriteActive := TRUE;
     16#32: // Write constant value
       #ArrayOutput[1] := 16#32;
       #PointerByte := #Offset_DBSend;
       #WriteActive := TRUE;
       #ShortCom := TRUE;
     16#81: // Read user data       
       #ArrayOutput[1] := 16#81;
       #PointerByte := #Offset_DBReceive;
       #ReadActive := TRUE;
     16#82: // Write user data       
       #ArrayOutput[1] := 16#82;
       #PointerByte := #Offset_DBSend;
       #WriteActive := TRUE;
     16#87: // Store Start address for Auto read
       #ArrayOutput[1] := 16#87;
       #WriteCom := TRUE;
     16#91: // Copy data between data carriers
       #ArrayOutput[1] := 16#91;
       #PointerByte := #Offset_DBReceive;
       #WriteCom := TRUE;
       #TotalByte := 0;
     16#92: // Initialize CRC16       
       #ArrayOutput[1] := 16#92;
       #PointerByte := #Offset_DBSend;
       #WriteActive := TRUE;
     16#B2: // Write constant value
       #ArrayOutput[1] := 16#B2;
       #PointerByte := #Offset_DBSend;
       #WriteActive := TRUE;
       #ShortCom := TRUE;
     ELSE
       #tError := w#16#81; // Error no com selected
       GOTO Error;
   END_CASE;

   // Initialization at comando start
   #BytePerPage := UDINT_TO_INT(#PIcount - 2);
   #FirstCycle := TRUE;
   #Ready := FALSE;
   #ErrorCode := 0;
   #Error := FALSE;
   #ErrorInt := FALSE;
   #tError := 0;
   #ToggleOld := #bHd_TO_ToggleOut;
   #BIS_STA.Ready := FALSE;
   #BIS_STA.Busy := TRUE;
   // Adding Command trailer

   IF #WriteCom THEN
     #TotalByte := 0;
   END_IF;
   // Command send -> set AV

   CASE #Command OF
     16#1, 16#2, 16#12: // User Commando
       #TotalByte := #TAG_NumbOfByte;
       #ArrayOutput[2] := DINT_TO_BYTE(#TAG_StartAddr);
       #ArrayOutput[3] := DINT_TO_BYTE(SHR(IN := #TAG_StartAddr, N := 8));
       #ArrayOutput[4] := DINT_TO_BYTE(#TAG_NumbOfByte);
       #ArrayOutput[5] := DINT_TO_BYTE(SHR(IN := #TAG_NumbOfByte, N := 8));
     16#7:// Auto read address
       #TotalByte := 0;
       #ArrayOutput[2] := DINT_TO_BYTE(#TAG_StartAddr);
       #ArrayOutput[3] := DINT_TO_BYTE(SHR(IN := #TAG_StartAddr, N := 8));
     16#9: // Read Typ and Serial  
       #ArrayOutput[1] := 16#9;
       #PointerByte := #Offset_DBReceive;
       #RdLengIn := TRUE;
       #ReadActive := TRUE;
     16#11: // Copy 
       #ArrayOutput[2] := DINT_TO_BYTE(#TAG_StartAddr);
       #ArrayOutput[3] := DINT_TO_BYTE(SHR(IN := #TAG_StartAddr, N := 8));
       #ArrayOutput[4] := DINT_TO_BYTE(#CopTargetAddr);
       #ArrayOutput[5] := DINT_TO_BYTE(SHR(IN := #CopTargetAddr, N := 8));
       #ArrayOutput[6] := DINT_TO_BYTE(#TAG_NumbOfByte);
       #ArrayOutput[7] := DINT_TO_BYTE(SHR(IN := #TAG_NumbOfByte, N := 8));
       #ArrayOutput[8] := INT_TO_BYTE(#CopRW_HeadNo);
     16#13, 16#14: // Read or Write DSFID overwrite unused bytes
       #ArrayOutput[2] := 0;
       #ArrayOutput[3] := 0;
       #ArrayOutput[4] := 0;
       #ArrayOutput[5] := 0;
     16#32: //Write constant
       IF (#IOLink_Proc OR #CLM_Proc) AND
         NOT #IOLink_Proc401 THEN // Only for IO Link
         #TotalByte := 0;
         #WriteCom := TRUE;
         IF IS_ARRAY(#DB_SendOpt) AND TypeOfElements(#DB_SendOpt) <> Byte THEN
           #tError := w#16#85; //Error read input data
           GOTO Error;

         ELSIF IS_ARRAY(#DB_SendOpt) AND TypeOfElements(#DB_SendOpt) = Byte THEN
           #RetValVarMove := MOVE_BLK_VARIANT(SRC := #DB_SendOpt,
                                              COUNT := 1,// 1 Byte for Copy
                                              SRC_INDEX := #PointerByte,
                                              DEST_INDEX := 6,
                                              DEST => #ArrayOutput);

           IF #RetValVarMove <> 0 THEN
             #tError := w#16#88; //Error read input data
             GOTO Error;
           END_IF;

         ELSE // DB Number Assigned

           #ArrayOutput[6] := PEEK(area := 16#84,
                                   dbNumber := #tempDB,
                                   byteOffset := #PointerByte);
         END_IF;

       ELSE
         #TotalByte := 1;
       END_IF;
       #ArrayOutput[2] := DINT_TO_BYTE(#TAG_StartAddr);
       #ArrayOutput[3] := DINT_TO_BYTE(SHR(IN := #TAG_StartAddr, N := 8));
       #ArrayOutput[4] := DINT_TO_BYTE(#TAG_NumbOfByte);
       #ArrayOutput[5] := DINT_TO_BYTE(SHR(IN := #TAG_NumbOfByte, N := 8));

     16#81, 16#82, 16#92:
       #TotalByte := #TAG_NumbOfByte;
       #ArrayOutput[2] := DINT_TO_BYTE(#TAG_StartAddr);
       #ArrayOutput[3] := DINT_TO_BYTE(SHR(IN := #TAG_StartAddr, N := 8));
       #ArrayOutput[4] := DINT_TO_BYTE(SHR(IN := #TAG_StartAddr, N := 16));
       #ArrayOutput[5] := DINT_TO_BYTE(#TAG_NumbOfByte);
       #ArrayOutput[6] := DINT_TO_BYTE(SHR(IN := #TAG_NumbOfByte, N := 8));
       #ArrayOutput[7] := DINT_TO_BYTE(SHR(IN := #TAG_NumbOfByte, N := 16));

     16#87:
       #TotalByte := 0;
       #ArrayOutput[2] := DINT_TO_BYTE(#TAG_StartAddr);
       #ArrayOutput[3] := DINT_TO_BYTE(SHR(IN := #TAG_StartAddr, N := 8));
       #ArrayOutput[4] := DINT_TO_BYTE(SHR(IN := #TAG_StartAddr, N := 16));
     16#91:
       #ArrayOutput[2] := DINT_TO_BYTE(#TAG_StartAddr);
       #ArrayOutput[3] := DINT_TO_BYTE(SHR(IN := #TAG_StartAddr, N := 8));
       #ArrayOutput[4] := DINT_TO_BYTE(SHR(IN := #TAG_StartAddr, N := 16));
       #ArrayOutput[5] := DINT_TO_BYTE(#CopTargetAddr);
       #ArrayOutput[6] := DINT_TO_BYTE(SHR(IN := #CopTargetAddr, N := 8));
       #ArrayOutput[7] := DINT_TO_BYTE(SHR(IN := #CopTargetAddr, N := 16));
       #ArrayOutput[8] := DINT_TO_BYTE(#TAG_NumbOfByte);
       #ArrayOutput[9] := DINT_TO_BYTE(SHR(IN := #TAG_NumbOfByte, N := 8));
       #ArrayOutput[10] := DINT_TO_BYTE(SHR(IN := #TAG_NumbOfByte, N := 16));
       #ArrayOutput[11] := INT_TO_BYTE(#CopRW_HeadNo);
     16#B2: //Write constant
       #TotalByte := 1;
       #ArrayOutput[2] := DINT_TO_BYTE(#TAG_StartAddr);
       #ArrayOutput[3] := DINT_TO_BYTE(SHR(IN := #TAG_StartAddr, N := 8));
       #ArrayOutput[4] := DINT_TO_BYTE(SHR(IN := #TAG_StartAddr, N := 16));
       #ArrayOutput[5] := DINT_TO_BYTE(#TAG_NumbOfByte);
       #ArrayOutput[6] := DINT_TO_BYTE(SHR(IN := #TAG_NumbOfByte, N := 8));
       #ArrayOutput[7] := DINT_TO_BYTE(SHR(IN := #TAG_NumbOfByte, N := 16));
   END_CASE;

   #bHd_AV_JobStart := TRUE;
   GOTO DataOut; // wite to output
   //-----------------------------------------------------------------------------
   // Read userdata or multi epc comand
   //----------------------------------------------------------------------------- 
   Read: ;

   IF NOT #bHd_AE_JobEnd AND
     #WaitOnAE OR
     #bHd_AF_JobError OR
     NOT #bHd_AA_JobStart THEN
     RETURN;
   END_IF;

   // Toggled?
   IF (NOT #FirstCycle OR NOT #WaitOnAE) AND
     ((#ToggleOld AND #bHd_TO_ToggleOut) OR
     (NOT #ToggleOld AND NOT #bHd_TO_ToggleOut))
   THEN
     RETURN;
   END_IF;

   IF #RdLengIn AND #FirstCycle THEN
     IF #ArrayInput[1] <= 64 THEN
       #TotalByte := #ArrayInput[1] + 1;
     ELSE
       #TotalByte := 0;
     END_IF;
   END_IF;

   #tempDB := #DB_Receive ;

   IF #TotalByte <= #BytePerPage THEN
     #LengthByte := #TotalByte;
   ELSE
     #LengthByte := #BytePerPage;
   END_IF;

   IF IS_ARRAY(#DB_ReceiveOpt) AND TypeOfElements(#DB_ReceiveOpt) <> Byte THEN
     #tError := w#16#85; //Error read input data
     GOTO Error;

   ELSIF IS_ARRAY(#DB_ReceiveOpt) AND TypeOfElements(#DB_ReceiveOpt) = Byte THEN
     #RetValVarMove := MOVE_BLK_VARIANT(SRC := #ArrayInput,
                                        COUNT := DINT_TO_UDINT(#LengthByte),
                                        SRC_INDEX := 1,
                                        DEST_INDEX := #PointerByte,
                                        DEST => #DB_ReceiveOpt);
     IF #RetValVarMove <> 0 THEN
       #tError := w#16#86; //Error read moveblock
       GOTO Error;
     END_IF;

   ELSE
     FOR #tLoop := 0 TO #LengthByte - 1 DO // Not Optimized
       POKE(area := 16#84,
            dbNumber := #tempDB,
            byteOffset := #PointerByte + #tLoop,
            value := #ArrayInput[1 + #tLoop]);
     END_FOR;
   END_IF;
   GOTO Com_End;
   //-----------------------------------------------------------------------------
   // Write comand
   //----------------------------------------------------------------------------- 
   Write: ;
   IF #bHd_AE_JobEnd THEN
     GOTO AV_Reset;
   END_IF;

   IF NOT #bHd_AA_JobStart OR
     #bHd_AF_JobError THEN
     RETURN;
   END_IF;

   IF ((#ToggleOld AND #bHd_TO_ToggleOut) OR
     (NOT #ToggleOld AND NOT #bHd_TO_ToggleOut)) THEN
     RETURN;
   END_IF;

   IF #TotalByte <= #BytePerPage THEN
     #LengthByte := #TotalByte;
   ELSE
     #LengthByte := #BytePerPage;
   END_IF;

   #tempDB := #DB_Send;
   IF #LengthByte > 0 THEN
     IF IS_ARRAY(#DB_SendOpt) AND TypeOfElements(#DB_SendOpt) <> Byte THEN
       #tError := w#16#87; //Error read input data
       GOTO Error;

     ELSIF IS_ARRAY(#DB_SendOpt) AND TypeOfElements(#DB_SendOpt) = Byte THEN
       #RetValVarMove := MOVE_BLK_VARIANT(SRC := #DB_SendOpt,
                                          COUNT := DINT_TO_UDINT(#LengthByte),
                                          SRC_INDEX := #PointerByte,
                                          DEST_INDEX := 1,
                                          DEST => #ArrayOutput);

       IF #RetValVarMove <> 0 THEN
         #tError := w#16#88; //Error read input data
         GOTO Error;
       END_IF;

     ELSE

       FOR #tLoop := 0 TO #LengthByte - 1 DO
         #ArrayOutput[1 + #tLoop] := PEEK(area := 16#84,
                                          dbNumber := #tempDB,
                                          byteOffset := #PointerByte + #tLoop);
       END_FOR;
     END_IF;
   END_IF;
   Com_End:;
   //-----------------------------------------------------------------------------
   // Command block end 
   //----------------------------------------------------------------------------- 
   #TotalByte := #TotalByte - #LengthByte;
   #PointerByte := #PointerByte + #LengthByte;
   #ToggleOld := #bHd_TO_ToggleOut;
   #bHd_TI_ToggleIn := NOT #bHd_TI_ToggleIn;

   WriteCom:;

   #FirstCycle := FALSE;

   IF #TotalByte > 0 THEN
     GOTO DataOut;//End;
   END_IF;

   IF NOT #bHd_AE_JobEnd THEN
     GOTO DataOut;//End;
   END_IF;

   AV_Reset: ; //Reset job
   #ReadActive := FALSE;
   #WriteActive := FALSE;
   #ShortCom := FALSE;
   #RdLengIn := FALSE;
   #WriteCom := FALSE;
   #WaitOnAE := FALSE;
   #ToggleOld := false;
   #bHd_AV_JobStart := FALSE;
   #bHd_GR_Default := FALSE;
   #bHd_KA_HeadOff := FALSE;
   #bHd_TI_ToggleIn := FALSE;

   DataOut: // Outbput bit header
   #ArrayOutput[0].%X0 := #bHd_AV_JobStart;
   #ArrayOutput[0].%X2 := #bHd_GR_Default;
   #ArrayOutput[0].%X4 := #bHd_HD_HeadSel;
   #ArrayOutput[0].%X5 := #bHd_KA_HeadOff;
   #ArrayOutput[0].%X6 := #bHd_TI_ToggleIn;
   #ArrayOutput[0].%X7 := #bHd_Cttp_TagType;
   #ArrayOutput[#PQcount - 1] := #ArrayOutput[0]; // Copy to 2.nd Bitstring
   //-----------------------------------------------------------------------------
   // cyclic write plc output to BIS input
   //-----------------------------------------------------------------------------

   IF #HW_Init THEN

     IF #CLM_Proc THEN
       #tLCnt := 0;
       FOR #tLoop := UDINT_TO_DINT(#PQaddr) TO UDINT_TO_DINT(#PQaddr + #PQcount - 1) DO
         POKE(area := 16#82,
              dbNumber := 0,
              byteOffset := #tLoop,
              value := #ArrayOutput[#tLCnt]);
         #tLCnt := #tLCnt + 1;
       END_FOR;

     ELSE
       #RetVal_WR_DP := DPWR_DAT(LADDR := #HW_LADDR, RECORD := #ArrayOutput);
     END_IF;
   END_IF;

   #RetVal_Get_ErrID := GET_ERR_ID();

   IF #RetVal_Get_ErrID <> 0
     AND NOT #Init
     AND NOT #ErrorInt THEN
     #tError := 16#53;
     GOTO Error;
   END_IF;

   RETURN;
   //-----------------------------------------------------------------------------
   // Error output
   //-----------------------------------------------------------------------------
   Error: ;
   #ErrorCode := #tError;
   #Ready := FALSE;
   #Error := TRUE;
   #ErrorInt := TRUE;
   #BIS_STA.Error := TRUE;

   GOTO AV_Reset;
END_FUNCTION_BLOCK

FUNCTION_BLOCK "BVS_Sensor"   // FB52, SCL
TITLE = BVS_ID
{ S7_Optimized_Access := 'TRUE' }
AUTHOR : PD-ILS
FAMILY : Balluff
VERSION : 1.1
// Functionblock for BVS ID and BVS VS.
// Compatible with Profinet and IO-Link version.
   VAR_INPUT
      Init : Bool;   // Internal reset and initailisation of FB
      CommandStart : Bool;   // Start BVS command
      BVS_ResetError : Bool;   // Reset BVS errors
      BVS_Trigger : Bool;   // Trigger BVS
      Get_Results : Bool;   // Get BVS results
      HW_LADDR : Hw_SubModule;   // BVS hardware address
      Command : Int;   // 1=SwitchApp; 2=GetApp; 3=GetResult; 4=SetInput
      DB_Send : Int;   // Data block with BVS send data
      Offset_DBSend : Int;   // Offset send data
      DB_Receive : Int;   // Data block with BVS receive data
      Offset_DBReceive : Int;   // Offset receive data
      Data_Length : Int;   // Data length for set commando
      WD_Time : Time := T#120000ms;   // Watchdog of commandos
      PILen : UInt := 32;   // Input process data length
      PQLen : UInt := 32;   // Output process data length
   END_VAR
   VAR_OUTPUT
      Ready : Bool;   // Comamnd ready and FB ready
      BVS_WaitForTrigger : Bool;   // BVS waiting for Trigger
      BVS_ResultDataAvailable : Bool;   // BVS result ready
      BVS_Ready : Bool;   // BVS ready
      BVS_DeviceLocked : Bool;   // BVS is locked
      BVS_TriggerOverflowError : Bool;   // BVS warning overtriggerd
      BVS_ResultDataError : Bool;   // BVS warning result data error
      BVS_ReportError : Bool;   // BVS warning report error
      BVS_InputDataError : Bool;   // BVS warning input data error
      BVS_SystemError : Bool;   // BVS warning system error
      Error : Bool;   // Command or BVS Error
      ErrorNumber : Word;   // Error number
      ReceivedLength : Int;   // BVS received result buffer length
   END_VAR
   VAR
      PointerByte : Int;   // Pointer byte
      LengthByte : Int;   // Number of byte for set/get commando
      BytePerPageIn : Int;   // User bytes per page Out
      BytePerPageOut : Int;   // User bytes per page In
      TotalByte : Int;   // Over all byte data to be set/get
      LengOverhead : Int;   // Overhead length for get command
      StDataOffset : Int;   // Start Data Offset for set command
      HW_Init : Bool;   // Hardware adresses initialized
      GetCommandActive : Bool;   // Get commado activ
      SetCommandActive : Bool;   // Set commando active
      GComSend : Bool;   // Get Commando send
      ComDatEnd : Bool;   // Comand data transfered
      ToggleOld : Bool;   // Toggle bit last cycle
      FirstCycle : Bool;   // First command cycle
      IMP_Start : Bool;   // Rising edge Start
      IMP_ResetError : Bool;   // Rising edge Reset
      Cam_Reset : Bool;   // Start BVS reset
      ErrorIn : Bool;   // Error bit intern
      WD_TimerIn : Bool;   // Watchdog timer input
      WD_TimerQ : Bool;   // Watchdog timer output
      CO_WaitForTrigger : Bool;   // CAM Out - PLC In waiting for trigger BasAd[50]
      CO_ResultDataAvailable : Bool;   // CAM Out - PLC In result ready
      CO_R02 : Bool;   // CAM Out - PLC In reserved
      CO_R03 : Bool;   // CAM Out - PLC In simulation mode activated
      CO_R04 : Bool;   // CAM Out - PLC In reserved
      CO_Ready : Bool;   // CAM Out - PLC In ready
      CO_R06 : Bool;   // CAM Out - PLC In reserved
      CO_DeviceLocked : Bool;   // CAM Out - PLC In device locked
      CO_TriggerOverflow : Bool;   // CAM Out - PLC In error trigger overflow
      CO_ResultDataError : Bool;   // CAM Out - PLC In result data overwitten
      CO_ReportError : Bool;   // CAM Out - PLC In ftp report error
      CO_R13 : Bool;   // CAM Out - PLC In reserved
      CO_InputDataError : Bool;   // CAM Out - PLC Input data error
      CO_R15 : Bool;   // CAM Out - PLC In reserved
      CO_R16 : Bool;   // CAM Out - PLC In reserved
      CO_SystemError : Bool;   // CAM Out - PLC In system error
      CO_R20 : Bool;   // CAM Out - PLC In reserved
      CO_JobStartAA : Bool;   // CAM Out - PLC In job start
      CO_JobEndAE : Bool;   // CAM Out - PLC In job end
      CO_JobErrorAF : Bool;   // CAM Out - PLC In job error
      CO_R24 : Bool;   // CAM Out - PLC In reserved
      CO_ToggleOut : Bool;   // CAM Out - PLC In toggle out
      CO_OutArea : Array[0..#OutBuSi] of Byte;   // CAM Out - PLC In data area
      CI_AV_JobStart : Bool;   // PLC Out - CAM In job start
      CI_Trigger : Bool;   // PLC Out - CAM In trigger
      CI_ResetError : Bool;   // PLC Out - CAM In reset error
      CI_R03 : Bool;   // PLC Out - CAM In reserved
      CI_R04 : Bool;   // PLC Out - CAM In reserved
      CI_R05 : Bool;   // PLC Out - CAM In reserved
      CI_ToggleIn : Bool;   // PLC Out - CAM In toggle in
      CI_R07 : Bool;   // PLC Out - CAM In reserved
      CI_InLengInt : Int;   // PLC Out - CAM In length int
      CI_InArea : Array[0..#InBuSi] of Byte;   // PLC Out - CAM In input area
      OldCyComState : Word;   // Commando state last cycle
      WD_Timer : TON_TIME;   // Watchdog timer TON
      PIaddr : UDInt;   // Input address
      PIcount : UInt;   // Input length
      PQaddr : UDInt;   // Output address
      PQcount : UInt;   // Output address
      RetVal_ModulDiag : Int;   // Return value modul diagnosis
      RetVal_RD_Addr : Int;   // Return value read address
      RetVal_RD_DP : Int;   // Return value read input data
      RetVal_WR_DP : Int;   // Return value write output data
      RetVal_Get_ErrID : Word;   // Return value get error ID
      R_TRIG_ResetError : R_TRIG;   // R Trigger reset warning
      R_TRIG_CamTrg : R_TRIG;   // R Trigger BVS trigger
      R_TRIG_Start : R_TRIG;   // R Trigger BVS start
      ErrorCode : DWord;   // Internal BVS error code
      CNT_Diag : UInt;   // CNT_Modul Diag
      Diag_Out : DWord;   // Modul Diag
   END_VAR
   VAR_TEMP
      tError : Word;   // temp error buffer
      tLoop : DInt;   // temp loopcounter
   END_VAR
   VAR CONSTANT
      InBuSi : Int := 127;   // maximum size input buffer
      OutBuSi : Int := 127;   // maximum size output buffer
      ST_DATOFFSET : Int := 3;   // First DataOffset for set commands
   END_VAR
BEGIN
   //=============================================================================
   //Balluff GmbH
   //(c)Copyright (2024) All Rights Reserved
   //-----------------------------------------------------------------------------
   //Library: BalluffVision
   //Tested with: CPU 1214C V4.1
   //Engineering: TIA Portal V13 SP1 
   //Restrictions: -
   //Requirements: PLC (S7-1200 / S7-1500)
   //Functionality: Boolean BVS functions, BVS Commandos
   //-----------------------------------------------------------------------------
   //Change log table:
   //Version  Date       Expert in charge      Changes applied
   //00.01.00 30.11.2022 Balluff GmbH PD-ILS   First created with TIA V13 SP1
   //00.01.10 30.01.2024 Balluff GmbH PD-ILS   FB name changed, buffer enlarged
   //=============================================================================
   //
   (*
   Disclaimer of Liability
   **********************
   The demo function block is free of charge and is a universal application 
   example.
   This demo function block shall help program and configure PLC applications and 
   shall provide possible solutions.
   The user is not entitled to claim for warranty, error correction and updates. 
   In 
   particular there is excluded any claims against Balluff GmbH for damages that 
   might result from the use of this demo program. Excluded from this limitation 
   of 
   liability shall be (a) those damages that are based on injury to life, limb or 
   health, (b) a liability according to the Produkthaftungsgesetz (German Product 
   Liability Law) and (c) cases of willful intent.
   Please check if the function block is intended for your application before 
   adapting it in plants and machineries.
   By using the S7 sample, made available free of charge you accept the limitation 
   of 
   warranty and liability!

   Haftungsausschluss:
   *********************
   Der hier kostenlos verfügbare DEMO-Baustein ist ein allgemeingültiges 
   Anwendungsbeispiel. Dieser DEMO-Baustein soll bei der Programmierung und 
   Projektierung von SPS-Anwendungen unterstützen und Lösungsansätze aufzeigen. 
   Ein Anspruch auf Gewährleistung, Fehlerbeseitigung und Update besteht für den 
   Anwender nicht. Die BALLUFF GmbH schließt insbesondere jegliche Haftung für 
   Schäden, die durch den Einsatz dieses DEMO-Bausteins entstehen, ausdrücklich 
   aus! Diese Haftungsbeschränkung gilt nicht bei Verletzungen des Lebens, des 
   Körpers oder der Gesundheit, bei der Haftung nach dem Produkthaftungsgesetz und 
   bei vorsätzlichen Pflichtverletzungen. 
   Prüfen Sie vor dem Einsatz in Anlagen und Maschinen, ob der hier 
   bereitgestellte 
   DEMO Baustein für Ihre Anwendung nutzbar ist!
   Mit dem Einsatz des hier kostenlos vorgelegten S7-Beispiel erkennen Sie die 
   Gewährleistungs- und Haftungsbegrenzung an!
   *)
   //-----------------------------------------------------------------------------
   //FB Init
   //-----------------------------------------------------------------------------
   IF #Init THEN
       #Ready := TRUE;
       #HW_Init := FALSE;
       #GetCommandActive := FALSE;
       #SetCommandActive := FALSE;
       #GComSend := FALSE;
       #ToggleOld := FALSE;
       #FirstCycle := FALSE;
       #ComDatEnd := False;
       #Error := FALSE;
       #ErrorIn := FALSE;
       #CI_AV_JobStart := FALSE;
       #CI_Trigger := FALSE;
       #CI_ResetError := false;
       #PointerByte := 0;
       #BytePerPageIn := 0;
       #BytePerPageOut := 0;
       #TotalByte := 0;
       #ReceivedLength := 0;
       #ErrorNumber := 0;
       #CO_OutArea[0] := 0;
       #CO_OutArea[1] := 0;
       #CO_OutArea[2] := 0;
       #BVS_Ready := FALSE;
   END_IF;
   //-----------------------------------------------------------------------------
   // Read modul states
   //-----------------------------------------------------------------------------
   #RetVal_ModulDiag := GET_DIAG(MODE := 0, LADDR := #HW_LADDR, CNT_DIAG => #CNT_Diag, DIAG := #Diag_Out);

   //-----------------------------------------------------------------------------
   // Reading PI/PQ addr and data length
   //-----------------------------------------------------------------------------
   IF NOT #HW_Init THEN
     #RetVal_RD_Addr := RD_ADDR(LADDR := #HW_LADDR , PIADDR => #PIaddr, PICount => #PIcount,
                                  PQADDR => #PQaddr, PQCount => #PQcount);
       #HW_Init := TRUE;
       // Overwrite PI and PO Lenght with lenth from FB input
       #PIcount := #PILen;
       #PQcount := #PQLen;
   END_IF;
   //-----------------------------------------------------------------------------
   // Cyclic read cam input if HW init done
   //----------------------------------------------------------------------------- 
   IF #HW_Init THEN
     #RetVal_RD_DP := DPRD_DAT(LADDR := #HW_LADDR, RECORD => #CO_OutArea);
   END_IF;

   IF #RetVal_RD_DP <> 0 THEN
     FOR  #tLoop := 0 TO #OutBuSi DO
       #CO_OutArea[#tLoop] := 0;
     END_FOR;
   END_IF;

   IF #Init THEN
     GOTO JobReset;
   END_IF;
   //-----------------------------------------------------------------------------
   // Move input bytes to static bits
   //  CO == Camera Outputs
   //-----------------------------------------------------------------------------
   // Byte 0 - Product Status Bits
   #CO_WaitForTrigger := #CO_OutArea[0].%X0;
   #CO_ResultDataAvailable := #CO_OutArea[0].%X1;
   #CO_R02 := #CO_OutArea[0].%X2;
   #CO_R03 := #CO_OutArea[0].%X3;
   #CO_R04 := #CO_OutArea[0].%X4;
   #CO_Ready := #CO_OutArea[0].%X5;
   #CO_R06 := #CO_OutArea[0].%X6;
   #CO_DeviceLocked := #CO_OutArea[0].%X7;
   //Byte 1 - Error Signals
   #CO_TriggerOverflow := #CO_OutArea[1].%X0;
   #CO_ResultDataError := #CO_OutArea[1].%X1;
   #CO_ReportError := #CO_OutArea[1].%X2;
   #CO_R13 := #CO_OutArea[1].%X3;
   #CO_InputDataError := #CO_OutArea[1].%X4;
   #CO_R15 := #CO_OutArea[1].%X5;
   #CO_R16 := #CO_OutArea[1].%X6;
   #CO_SystemError := #CO_OutArea[1].%X7;

   //-----------------------------------------------------------------------------
   // Move status-/warnbits to FB output 
   //-----------------------------------------------------------------------------
   #BVS_ResultDataAvailable := #CO_ResultDataAvailable;
   #BVS_WaitForTrigger := #CO_WaitForTrigger;
   #BVS_Ready := #CO_Ready;
   #BVS_DeviceLocked := #CO_DeviceLocked;
   #BVS_TriggerOverflowError := #CO_TriggerOverflow;
   #BVS_ResultDataError := #CO_ResultDataError;
   #BVS_ReportError := #CO_ReportError;
   #BVS_InputDataError := #CO_InputDataError;
   #BVS_SystemError := #CO_SystemError;

   //-----------------------------------------------------------------------------
   // Comapre bitheader
   //-----------------------------------------------------------------------------
   IF #CO_OutArea[2] <> #CO_OutArea[#PIcount - 1] THEN
     RETURN;
   END_IF;
   //Byte 2 - Bit Header
   #CO_R20 := #CO_OutArea[2].%X0;
   #CO_JobStartAA := #CO_OutArea[2].%X1;
   #CO_JobEndAE := #CO_OutArea[2].%X2;
   #CO_JobErrorAF := #CO_OutArea[2].%X3;
   #CO_ToggleOut := #CO_OutArea[2].%X5;

   //-----------------------------------------------------------------------------
   // Check camera error bit
   //-----------------------------------------------------------------------------
   IF #CO_JobErrorAF AND NOT #ErrorIn THEN
     #tError := #CO_OutArea[3];
     GOTO Error;
   END_IF;

   //-----------------------------------------------------------------------------
   // Reset camera errors
   //-----------------------------------------------------------------------------
   #R_TRIG_ResetError(CLK:=#BVS_ResetError,
                   Q=>#IMP_ResetError);
   IF #IMP_ResetError THEN
       #Error := FALSE;
       #ErrorIn := FALSE;
       #ErrorNumber := 0;
       #CI_ResetError := TRUE;
   END_IF;

   IF NOT #BVS_ResetError
     THEN
       #CI_ResetError := FALSE;
   END_IF;

   //-----------------------------------------------------------------------------
   // Control boolean camera signals
   //-----------------------------------------------------------------------------
   #R_TRIG_CamTrg(CLK:=#BVS_Trigger);

   IF #R_TRIG_CamTrg.Q THEN
     #CI_Trigger := TRUE;
   END_IF;

   IF  NOT #BVS_Trigger THEN
     #CI_Trigger := FALSE;
   END_IF;

   //-----------------------------------------------------------------------------
   // Move  FB input to processdata output
   //-----------------------------------------------------------------------------
   #CI_InArea[0].%X0 := #CI_AV_JobStart;
   #CI_InArea[0].%X1 := #CI_Trigger;
   #CI_InArea[0].%X2 := #CI_ResetError;
   #CI_InArea[0].%X6 := #CI_ToggleIn;

   //-----------------------------------------------------------------------------
   // FB ready output 
   #Ready := ( #BVS_Ready 
             AND NOT #GetCommandActive 
             AND NOT #SetCommandActive 
             AND NOT #CO_JobStartAA 
             AND NOT #CO_JobEndAE);

   //-----------------------------------------------------------------------------
   // Command Start
              #R_TRIG_Start(CLK := #CommandStart OR #Get_Results,
                 Q => #IMP_Start);

   //-----------------------------------------------------------------------------
   // Generate error timeout
   //-----------------------------------------------------------------------------
   #WD_TimerIn := #SetCommandActive OR #GetCommandActive;

   #WD_Timer(IN := #WD_TimerIn,
             PT := #WD_Time,
             Q => #WD_TimerQ);

   IF #WD_TimerQ THEN
       #tError := w#16#30;
       GOTO Error;
   END_IF;

   //-----------------------------------------------------------------------------
   // Check HW/Profinet Error when start is set
   //-----------------------------------------------------------------------------
   IF #IMP_Start THEN
     IF #RetVal_RD_Addr <> 0 THEN
       #tError := w#16#40; //Error read address
       GOTO Error;
     END_IF;

     IF #RetVal_RD_DP <> 0 THEN
       #tError := w#16#41; //Error read input data
       GOTO Error;
     END_IF;

     IF #RetVal_WR_DP <> 0 THEN
       #tError := w#16#42; //Error read output data
       GOTO Error;
     END_IF;
   END_IF;

   //-----------------------------------------------------------------------------
   // Generate error data length
   //-----------------------------------------------------------------------------
   IF #IMP_Start AND
       (#Data_Length < 0) THEN
       #tError := w#16#32;
       GOTO Error;
   END_IF;

   //-----------------------------------------------------------------------------
   // Check controll- bits change - data output
   //-----------------------------------------------------------------------------
   IF #CI_InArea[0] <> #OldCyComState AND NOT #IMP_Start THEN
     GOTO DataOutput;
   END_IF;
   //=============================================================================
   //
   // Camera commandos
   //
   //=============================================================================

   //-----------------------------------------------------------------------------
   // Goto FB end if no job active
   //-----------------------------------------------------------------------------
   IF (NOT #GetCommandActive AND
       NOT #SetCommandActive AND
      (NOT #IMP_Start OR NOT #Ready)) THEN 
       RETURN;
   END_IF;

   IF #ComDatEnd THEN  // Check Get or Set
     GOTO CheckHsAck; //CommandEnd;
   ELSIF #GetCommandActive THEN
     GOTO GetCommand;
   ELSIF #SetCommandActive THEN
     GOTO SetCommand;
   END_IF;

   //-----------------------------------------------------------------------------
   // Initialize Command
   //-----------------------------------------------------------------------------
   #CI_InArea[2] := 0;
   #CI_InArea[3] := 0;

   IF #Get_Results THEN
     #GetCommandActive := TRUE;
     #CI_InArea[1] := 3;
     #CI_InLengInt := 0;
     #LengOverhead := 3;
   ELSE

     CASE #Command OF
       1: // Switch Application
         #SetCommandActive := TRUE;
         #CI_InArea[1] := 1;
         #TotalByte := 4;
         #CI_InLengInt := 4;
       2:  // Get Application ID
         #GetCommandActive := TRUE;
         #CI_InArea[1] := 2;
         #CI_InLengInt := 0;
         #LengOverhead := 3;
       3:  // Get Results
         #GetCommandActive := TRUE;
         #CI_InArea[1] := 3;
         #CI_InLengInt := 0;
         #LengOverhead := 3;
       4:  // Set Inputs       
         #SetCommandActive := TRUE;
         #CI_InArea[1] := 4;
         #TotalByte := #Data_Length;
         #CI_InLengInt := #Data_Length;
       6:  // Get Date and Time 
         #GetCommandActive := TRUE;
         #CI_InArea[1] := 6;
         #CI_InLengInt := 0;
         #LengOverhead := 3;
       7:  // Set Date and Time      
         #SetCommandActive := TRUE;
         #CI_InArea[1] := 7;
         #TotalByte := 7 + #ST_DATOFFSET;
         #CI_InLengInt := 7;
       ELSE
         #tError := w#16#31;
         GOTO Error;
     END_CASE;
   END_IF;

   //-----------------------------------------------------------------------------
   // At 1st command step:
   // Calculate transmission data length fix bytes + bitheader
   // Delete output signals
   // Notice TO Bit
   //-----------------------------------------------------------------------------
   #BytePerPageIn := UDINT_TO_INT(#PIcount - 4);
   #BytePerPageOut := UDINT_TO_INT(#PQcount - 2);

   #FirstCycle := TRUE;
   #Ready := FALSE;
   #ErrorNumber := 0;
   #Error := FALSE;
   #ErrorIn := FALSE;
   #tError := 0;
   #GComSend := FALSE;
   #ReceivedLength := 0;
   #ToggleOld := #CO_ToggleOut;
   #CI_AV_JobStart := TRUE;

   IF NOT #SetCommandActive THEN
       GOTO GetCommand;
   END_IF;

   //-----------------------------------------------------------------------------
   // Set command, move data from "DB_Send" to camera
   //-----------------------------------------------------------------------------
   SetCommand: ;

   IF NOT #FirstCycle  
       AND ((#ToggleOld AND #CO_ToggleOut)
       OR (NOT #ToggleOld AND NOT #CO_ToggleOut)
       OR  NOT #CO_JobStartAA)
     THEN
       RETURN;
   END_IF;

   IF #FirstCycle THEN
     #PointerByte := #Offset_DBSend;
     #StDataOffset := #ST_DATOFFSET;
     #CI_InArea[2] := INT_TO_BYTE(SHR(IN := #CI_InLengInt, N := 8)); 
     #CI_InArea[3] := INT_TO_BYTE(#CI_InLengInt); 
   END_IF;

   IF #TotalByte <= #BytePerPageOut - #StDataOffset THEN
     #LengthByte := #TotalByte;
   ELSE
     #LengthByte := #BytePerPageOut - #StDataOffset;
   END_IF;

   FOR #tLoop := 0 TO #LengthByte - 1 DO 
     #CI_InArea[1 + #tLoop + #StDataOffset] := PEEK(area := 16#84,
                                      dbNumber := #DB_Send,
                                      byteOffset := #PointerByte + #tLoop);
     END_FOR;

   GOTO CommandEnd;

   GetCommand:;
   //-----------------------------------------------------------------------------
   // Get command
   // Send get commando goto Data output in first cycle 
   // 
   //-----------------------------------------------------------------------------
   IF #FirstCycle AND NOT #GComSend THEN
     #GComSend := TRUE;
     GOTO DataOutput;
   END_IF;

   IF #FirstCycle AND #CI_InArea[1] <> #CO_OutArea[3] // Check result code at 1st cycl 
     AND NOT #CO_JobStartAA
     OR NOT #CO_JobEndAE 
   THEN
     RETURN;
   END_IF;

   IF NOT #FirstCycle
     AND ((#ToggleOld AND #CO_ToggleOut)
     OR (NOT #ToggleOld AND NOT #CO_ToggleOut))
   THEN
     RETURN;
   END_IF;

   //-----------------------------------------------------------------------------
   // Read camera length byte at 1st cycle
   // move data from camera to "DB_Receive"
   //  
   //----------------------------------------------------------------------------- 
   IF #FirstCycle THEN

     #TotalByte := BYTE_TO_INT(#CO_OutArea[5]) +
     SHL(IN := BYTE_TO_INT(#CO_OutArea[4]), N := 8)+
     #LengOverhead;

     #PointerByte := #Offset_DBReceive;

     IF (#TotalByte < 0) THEN
       #tError := 16#32;
       GOTO Error;
     END_IF;

     #ReceivedLength := #TotalByte;

   END_IF; // End_IF First Cycle

   IF #TotalByte <= #BytePerPageIn THEN
     #LengthByte := #TotalByte;
    ELSE
     #LengthByte := #BytePerPageIn;
   END_IF;

   FOR #tLoop := 0 TO #LengthByte - 1 DO
     POKE(area := 16#84,
          dbNumber := #DB_Receive,
          byteOffset := #PointerByte + #tLoop,
          value := #CO_OutArea[3 + #tLoop]);
   END_FOR;

   CommandEnd:;

   //-----------------------------------------------------------------------------
   // Get and Set Command End
   //----------------------------------------------------------------------------- 
   IF NOT #ComDatEnd THEN
     #TotalByte := #TotalByte - #LengthByte;
     #PointerByte := #PointerByte + #LengthByte;
   END_IF;

   IF #TotalByte <= 0 THEN
     #ComDatEnd := TRUE;
   END_IF;

   IF (#GetCommandActive AND NOT #ComDatEnd) OR
     (NOT #FirstCycle AND #SetCommandActive) THEN
     #CI_ToggleIn := NOT #CI_ToggleIn;
   END_IF;

   #ToggleOld := #CO_ToggleOut;
   #FirstCycle := FALSE;
   #StDataOffset := 0;
   CheckHsAck:;

   IF (#CO_JobStartAA AND #CO_JobEndAE AND #ComDatEnd) THEN 
       #ComDatEnd := FALSE;
       #GetCommandActive := FALSE;
       #SetCommandActive := FALSE;
       #CI_AV_JobStart := FALSE;
       #CI_ToggleIn := FALSE;
       #ToggleOld := FALSE;
   END_IF;

   //-----------------------------------------------------------------------------
   // Data output fieldbus
   //-----------------------------------------------------------------------------
   DataOutput:;
   // Move bits to byte
   #CI_InArea[0].%X0 := #CI_AV_JobStart;
   #CI_InArea[0].%X1 := #CI_Trigger;
   #CI_InArea[0].%X2 := #CI_ResetError;
   #CI_InArea[0].%X6 := #CI_ToggleIn ;
   #CI_InArea[#PQcount - 1] := #CI_InArea[0];
   #OldCyComState := #CI_InArea[0];

   //-----------------------------------------------------------------------------
   // cyclic write plc output to cam input
   //-----------------------------------------------------------------------------
   IF #HW_Init  THEN
     #RetVal_WR_DP := DPWR_DAT(LADDR := #HW_LADDR, RECORD := #CI_InArea);
   END_IF;
   #RetVal_Get_ErrID := GET_ERR_ID();

   IF #RetVal_Get_ErrID <> 0
     AND NOT #Init
     AND NOT #ErrorIn THEN
     #tError := 16#43;
     GOTO Error;
   END_IF;

   RETURN; // FB End
   //-----------------------------------------------------------------------------
   // Error output
   //-----------------------------------------------------------------------------
   Error: ;
     #ErrorNumber := #tError;
     #Ready := FALSE;
     #Error := TRUE;
     #ErrorIn := TRUE;

   JobReset: ;
     #GetCommandActive := FALSE;
     #SetCommandActive := FALSE;
     #CI_AV_JobStart := FALSE;
     #CI_ToggleIn := FALSE;
     #ComDatEnd := FALSE;
     #ToggleOld := FALSE;
     GOTO DataOutput;
END_FUNCTION_BLOCK

ORGANIZATION_BLOCK "Main"   // OB1, LAD, ProgramCycle
TITLE = "Main Program Sweep (Cycle)"
{ S7_Optimized_Access := 'TRUE' }
VERSION : 0.1
   VAR_INPUT
      Initial_Call : Bool;   // Initial call of this OB
      Remanence : Bool;   // =True, if remanent data are available
   END_VAR
BEGIN

REGION Network 1 (SCL): kod stanowisko1 rfid
   IF "RFID1" AND "DB_Data".Stanowisko1.Sensors.RFID.CmdRead THEN
       "BIS_V_CLM_COM_DB_2".Command := 1;
       "BIS_V_CLM_COM_DB_2".TAG_StartAddr := 8;
       "BIS_V_CLM_COM_DB_2".TAG_NumbOfByte := 3;
       "BIS_V_CLM_COM_DB_2".Start := TRUE;

   ELSIF "RFID1" AND "DB_Data".Stanowisko1.Sensors.RFID.CmdWrite THEN
       "BIS_V_CLM_COM_DB_2".Command := 2;
       "BIS_V_CLM_COM_DB_2".TAG_StartAddr := 8;
       "BIS_V_CLM_COM_DB_2".TAG_NumbOfByte := 3;
       "BIS_V_CLM_COM_DB_2".Start := TRUE;

   ELSE
       // Jeśli nie ma komend, ściągamy Start na FALSE
       "BIS_V_CLM_COM_DB_2".Start := FALSE;
   END_IF;
END_REGION

REGION Network 2: blok stanowisko1 rfid
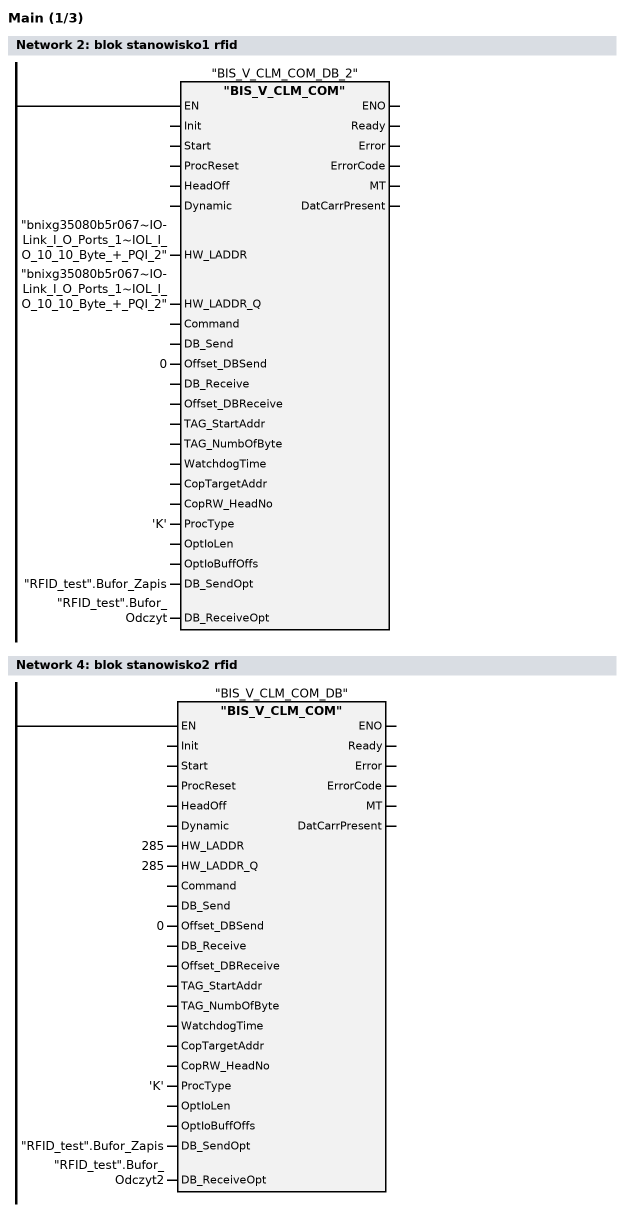
   RUNG wire#powerrail
      "BIS_V_CLM_COM_DB_2"(Init :=, Start :=, ProcReset :=, HeadOff :=, Dynamic :=, HW_LADDR := "bnixg35080b5r067~IO-Link_I_O_Ports_1~IOL_I_O_10_10_Byte_+_PQI_2", HW_LADDR_Q := "bnixg35080b5r067~IO-Link_I_O_Ports_1~IOL_I_O_10_10_Byte_+_PQI_2", Command :=, DB_Send :=, Offset_DBSend := 0, DB_Receive :=, Offset_DBReceive :=, TAG_StartAddr :=, TAG_NumbOfByte :=, WatchdogTime :=, CopTargetAddr :=, CopRW_HeadNo :=, ProcType := 'K', OptIoLen :=, OptIoBuffOffs :=, DB_SendOpt := "RFID_test".Bufor_Zapis, DB_ReceiveOpt := "RFID_test".Bufor_Odczyt, Ready =>, Error =>, ErrorCode =>, MT =>, DatCarrPresent =>)
   END_RUNG
   // the same network as SCL:
   "BIS_V_CLM_COM_DB_2"(HW_LADDR := "bnixg35080b5r067~IO-Link_I_O_Ports_1~IOL_I_O_10_10_Byte_+_PQI_2",   // "BIS_V_CLM_COM"
                        HW_LADDR_Q := "bnixg35080b5r067~IO-Link_I_O_Ports_1~IOL_I_O_10_10_Byte_+_PQI_2",
                        Offset_DBSend := 0,
                        ProcType := 'K',
                        DB_SendOpt := "RFID_test".Bufor_Zapis,
                        DB_ReceiveOpt := "RFID_test".Bufor_Odczyt);
END_REGION

REGION Network 3 (SCL): kod stanowisko2 rfid
   IF "RFID2" AND "DB_Data".Stanowisko2.Sensors.RFID.CmdRead THEN
       "BIS_V_CLM_COM_DB".Command := 1;
       "BIS_V_CLM_COM_DB".TAG_StartAddr := 8;
       "BIS_V_CLM_COM_DB".TAG_NumbOfByte := 3;
       "BIS_V_CLM_COM_DB".Start := TRUE;

   ELSE
       // Jeśli nie ma komend, ściągamy Start na FALSE
       "BIS_V_CLM_COM_DB".Start := FALSE;
   END_IF;
END_REGION

REGION Network 4: blok stanowisko2 rfid
   RUNG wire#powerrail
      "BIS_V_CLM_COM_DB"(Init :=, Start :=, ProcReset :=, HeadOff :=, Dynamic :=, HW_LADDR := 285, HW_LADDR_Q := 285, Command :=, DB_Send :=, Offset_DBSend := 0, DB_Receive :=, Offset_DBReceive :=, TAG_StartAddr :=, TAG_NumbOfByte :=, WatchdogTime :=, CopTargetAddr :=, CopRW_HeadNo :=, ProcType := 'K', OptIoLen :=, OptIoBuffOffs :=, DB_SendOpt := "RFID_test".Bufor_Zapis, DB_ReceiveOpt := "RFID_test".Bufor_Odczyt2, Ready =>, Error =>, ErrorCode =>, MT =>, DatCarrPresent =>)
   END_RUNG
   // the same network as SCL:
   "BIS_V_CLM_COM_DB"(HW_LADDR := 285,   // "BIS_V_CLM_COM"
                      HW_LADDR_Q := 285,
                      Offset_DBSend := 0,
                      ProcType := 'K',
                      DB_SendOpt := "RFID_test".Bufor_Zapis,
                      DB_ReceiveOpt := "RFID_test".Bufor_Odczyt2);
END_REGION

REGION Network 5 (SCL): kod stanowisko3 rfid
   IF "RFID3" AND "DB_Data".Stanowisko3.Sensors.RFID.CmdRead THEN
       "BIS_V_CLM_COM_DB_1".Command := 1;
       "BIS_V_CLM_COM_DB_1".TAG_StartAddr := 8;
       "BIS_V_CLM_COM_DB_1".TAG_NumbOfByte := 3;
       "BIS_V_CLM_COM_DB_1".Start := TRUE;

   ELSE
       // Jeśli nie ma komend, ściągamy Start na FALSE
       "BIS_V_CLM_COM_DB_1".Start := FALSE;
   END_IF;
END_REGION

REGION Network 6: blok stanowisko3 rfid
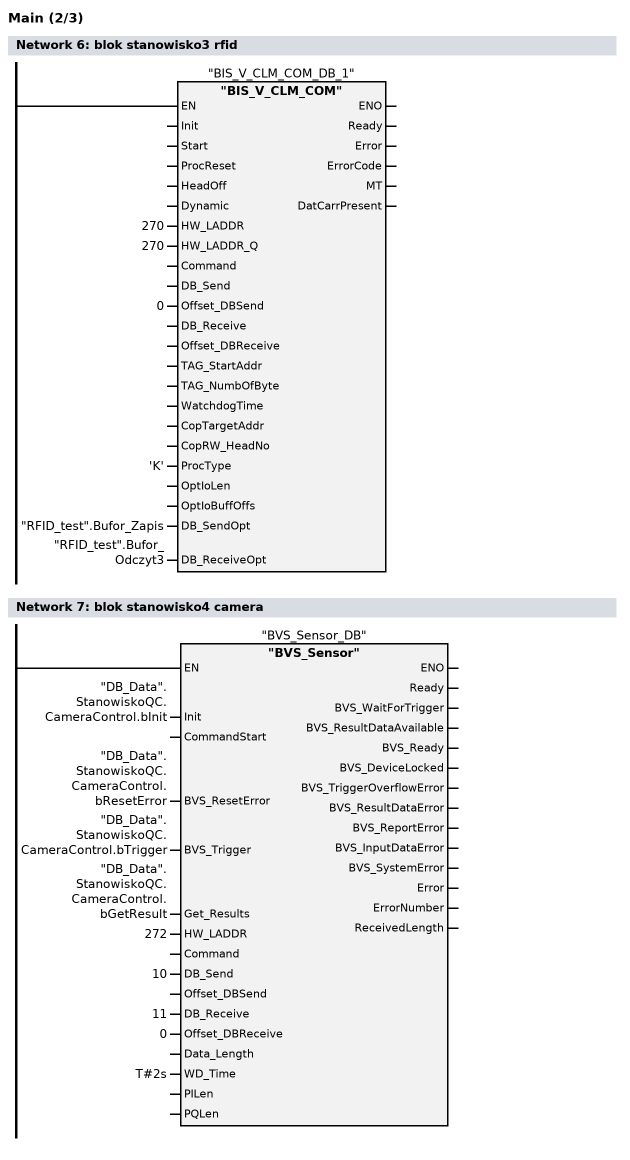
   RUNG wire#powerrail
      "BIS_V_CLM_COM_DB_1"(Init :=, Start :=, ProcReset :=, HeadOff :=, Dynamic :=, HW_LADDR := 270, HW_LADDR_Q := 270, Command :=, DB_Send :=, Offset_DBSend := 0, DB_Receive :=, Offset_DBReceive :=, TAG_StartAddr :=, TAG_NumbOfByte :=, WatchdogTime :=, CopTargetAddr :=, CopRW_HeadNo :=, ProcType := 'K', OptIoLen :=, OptIoBuffOffs :=, DB_SendOpt := "RFID_test".Bufor_Zapis, DB_ReceiveOpt := "RFID_test".Bufor_Odczyt3, Ready =>, Error =>, ErrorCode =>, MT =>, DatCarrPresent =>)
   END_RUNG
   // the same network as SCL:
   "BIS_V_CLM_COM_DB_1"(HW_LADDR := 270,   // "BIS_V_CLM_COM"
                        HW_LADDR_Q := 270,
                        Offset_DBSend := 0,
                        ProcType := 'K',
                        DB_SendOpt := "RFID_test".Bufor_Zapis,
                        DB_ReceiveOpt := "RFID_test".Bufor_Odczyt3);
END_REGION

REGION Network 7: blok stanowisko4 camera
   RUNG wire#powerrail
      "BVS_Sensor_DB"(Init := "DB_Data".StanowiskoQC.CameraControl.bInit, CommandStart :=, BVS_ResetError := "DB_Data".StanowiskoQC.CameraControl.bResetError, BVS_Trigger := "DB_Data".StanowiskoQC.CameraControl.bTrigger, Get_Results := "DB_Data".StanowiskoQC.CameraControl.bGetResult, HW_LADDR := 272, Command :=, DB_Send := 10, Offset_DBSend :=, DB_Receive := 11, Offset_DBReceive := 0, Data_Length :=, WD_Time := T#2s, PILen :=, PQLen :=, Ready =>, BVS_WaitForTrigger =>, BVS_ResultDataAvailable =>, BVS_Ready =>, BVS_DeviceLocked =>, BVS_TriggerOverflowError =>, BVS_ResultDataError =>, BVS_ReportError =>, BVS_InputDataError =>, BVS_SystemError =>, Error =>, ErrorNumber =>, ReceivedLength =>)
   END_RUNG
   // the same network as SCL:
   "BVS_Sensor_DB"(Init := "DB_Data".StanowiskoQC.CameraControl.bInit,   // "BVS_Sensor"
                   BVS_ResetError := "DB_Data".StanowiskoQC.CameraControl.bResetError,
                   BVS_Trigger := "DB_Data".StanowiskoQC.CameraControl.bTrigger,
                   Get_Results := "DB_Data".StanowiskoQC.CameraControl.bGetResult,
                   HW_LADDR := 272,
                   DB_Send := 10,
                   DB_Receive := 11,
                   Offset_DBReceive := 0,
                   WD_Time := T#2s);
END_REGION

REGION Network 8 (SCL)
   "DB_Data".StanowiskoQC.CameraControl.bInit := FALSE;
   "DB_Data".StanowiskoQC.CameraControl.CameraStatus := "BVS_Sensor_DB".BVS_Ready;


   CASE "DB_Data".StanowiskoQC.CameraControl.krok OF
       0:  // żądanie inspekcji -> najpierw wyczyść stary wynik jeśli wisi
           "DB_Data".StanowiskoQC.CameraControl.bTrigger := FALSE;
           "DB_Data".StanowiskoQC.CameraControl.bGetResult := FALSE;
           IF "DB_Data".StanowiskoQC.CameraControl.bZrobInspekcje
               AND "BVS_Sensor_DB".BVS_Ready THEN
               IF "BVS_Sensor_DB".BVS_ResultDataAvailable THEN
                   "DB_Data".StanowiskoQC.CameraControl.bGetResult := TRUE;  // skonsumuj stary
                   "DB_Data".StanowiskoQC.CameraControl.krok := 5;
               ELSE
                   "DB_Data".StanowiskoQC.CameraControl.krok := 8;           // nic nie wisi -> triggeruj
               END_IF;
           END_IF;

       5:  // czekaj aż flush ruszy
           IF NOT "BVS_Sensor_DB".Ready THEN
               "DB_Data".StanowiskoQC.CameraControl.krok := 6;
           END_IF;

       6:  // flush zakończony
           IF "BVS_Sensor_DB".Ready THEN
               "DB_Data".StanowiskoQC.CameraControl.bGetResult := FALSE;
               "DB_Data".StanowiskoQC.CameraControl.krok := 8;
           END_IF;

       8:  // wyzwól ŚWIEŻĄ inspekcję
           IF "BVS_Sensor_DB".BVS_WaitForTrigger THEN
               "DB_Data".StanowiskoQC.CameraControl.bTrigger := TRUE;
               "DB_Data".StanowiskoQC.CameraControl.krok := 10;
           END_IF;

       10:  // teraz ResultDataAvailable = ŚWIEŻY wynik
           "DB_Data".StanowiskoQC.CameraControl.bTrigger := FALSE;
           IF "BVS_Sensor_DB".BVS_ResultDataAvailable THEN
               "DB_Data".StanowiskoQC.CameraControl.bGetResult := TRUE;
               "DB_Data".StanowiskoQC.CameraControl.krok := 20;
           END_IF;

       20:  // czekaj aż FB ruszy z pobieraniem
           IF NOT "BVS_Sensor_DB".Ready THEN
               "DB_Data".StanowiskoQC.CameraControl.krok := 30;
           END_IF;

       30:  // dane pobrane -> NAJPIERW przepisz, POTEM skasuj
           IF "BVS_Sensor_DB".Ready THEN
               "DB_Data".StanowiskoQC.CameraControl.wynikOV[0] := ("DB_Cam_Output".Output[7] <> 0);
               "DB_Data".StanowiskoQC.CameraControl.wynikOV[1] := ("DB_Cam_Output".Output[8] <> 0);
               "DB_Data".StanowiskoQC.CameraControl.wynikOV[2] := ("DB_Cam_Output".Output[9] <> 0);
               "DB_Data".StanowiskoQC.CameraControl.wynikOV[3] := ("DB_Cam_Output".Output[10] <> 0);
               "DB_Data".StanowiskoQC.CameraControl.wynikOV[4] := ("DB_Cam_Output".Output[11] <> 0);
               "DB_Data".StanowiskoQC.CameraControl.wynikOV[5] := ("DB_Cam_Output".Output[12] <> 0);
               "DB_Data".StanowiskoQC.CameraControl.bGetResult := FALSE;
               "DB_Data".StanowiskoQC.CameraControl.bZrobInspekcje := FALSE;
               "DB_Data".StanowiskoQC.CameraControl.krok := 0;
           END_IF;
   END_CASE;
END_REGION

REGION Network 9
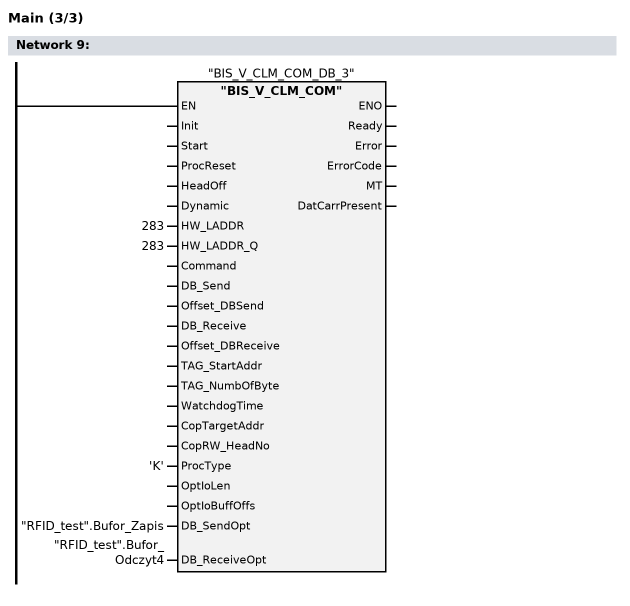
   RUNG wire#powerrail
      "BIS_V_CLM_COM_DB_3"(Init :=, Start :=, ProcReset :=, HeadOff :=, Dynamic :=, HW_LADDR := 283, HW_LADDR_Q := 283, Command :=, DB_Send :=, Offset_DBSend :=, DB_Receive :=, Offset_DBReceive :=, TAG_StartAddr :=, TAG_NumbOfByte :=, WatchdogTime :=, CopTargetAddr :=, CopRW_HeadNo :=, ProcType := 'K', OptIoLen :=, OptIoBuffOffs :=, DB_SendOpt := "RFID_test".Bufor_Zapis, DB_ReceiveOpt := "RFID_test".Bufor_Odczyt4, Ready =>, Error =>, ErrorCode =>, MT =>, DatCarrPresent =>)
   END_RUNG
   // the same network as SCL:
   "BIS_V_CLM_COM_DB_3"(HW_LADDR := 283,   // "BIS_V_CLM_COM"
                        HW_LADDR_Q := 283,
                        ProcType := 'K',
                        DB_SendOpt := "RFID_test".Bufor_Zapis,
                        DB_ReceiveOpt := "RFID_test".Bufor_Odczyt4);
END_REGION

REGION Network 10 (SCL): RFID4
   IF "RFID4" AND "DB_Data".StanowiskoQC.Sensors.RFID.CmdRead THEN
       "BIS_V_CLM_COM_DB_3".Command := 1;
       "BIS_V_CLM_COM_DB_3".TAG_StartAddr := 8;
       "BIS_V_CLM_COM_DB_3".TAG_NumbOfByte := 3;
       "BIS_V_CLM_COM_DB_3".Start := TRUE;

   ELSE
       // Jeśli nie ma komend, ściągamy Start na FALSE
       "BIS_V_CLM_COM_DB_3".Start := FALSE;
   END_IF;
END_REGION
END_ORGANIZATION_BLOCK

ORGANIZATION_BLOCK "Startup"   // OB100, SCL, Startup
TITLE = "Complete Restart"
{ S7_Optimized_Access := 'TRUE' }
VERSION : 0.1
   VAR_INPUT
      LostRetentive : Bool;   // True if retentive data are lost
      LostRTC : Bool;   // True if date and time are lost
   END_VAR
BEGIN
   "DB_Data".StanowiskoQC.CameraControl.bInit := TRUE;
END_ORGANIZATION_BLOCK

ORGANIZATION_BLOCK "Stanowisko1"   // OB123, SCL, ProgramCycle
TITLE = "Main Program Sweep (Cycle)"
{ S7_Optimized_Access := 'TRUE' }
VERSION : 0.1
   VAR_INPUT
      Initial_Call : Bool;   // Initial call of this OB
      Remanence : Bool;   // =True, if remanent data are available
   END_VAR
   VAR_TEMP
      temp_start_time : Int;
      temp_taget_time : Int;
      i : Int;
      Czas_DTL : DTL;
      Status_Czasu : Int;
      Minuty : Int;
      Sekundy : Int;
      StrMin : String;
      StrSec : String;
      temp_diff_time : Time;
   END_VAR
BEGIN
   // ===================== STANOWISKO 1 =====================
   CASE "DB_Data".Stanowisko1.Production.State OF

       0:
           //Ustawienie przyciskow
           "DB_Data".Stanowisko1.Commands.AbortProcess.Enable := 0;
           "DB_Data".Stanowisko1.Commands.FInish.Enable := 0;
           "DB_Data".Stanowisko1.Commands.ReportFault.Enable := 0;

           //Wyzerowanie stanu przyciskow (na wypadek zaleglych klikniec)
           "DB_Data".Stanowisko1.Commands.FInish.State := 0;
           "DB_Data".Stanowisko1.Commands.ReportFault.State := 0;

           //Ustawienie awarii na 0
           "DB_Data".Stanowisko1.Commands.FaultReason.DamagedPart := 0;
           "DB_Data".Stanowisko1.Commands.FaultReason.MissingPart := 0;
           "DB_Data".Stanowisko1.Commands.FaultReason.Other := 0;
           "DB_Data".Stanowisko1.Commands.FaultReason.PalletFault := 0;
           "DB_Data".Stanowisko1.Commands.FaultReason.SensorFault := 0;
           "DB_Data".Stanowisko1.Commands.FaultReason.WrongInstruction := 0;

           //Reset czasu cyklu na wyswietlaczu
           "DB_Data".Stanowisko1."Time".RemainingStr := '00:00';

           //Reset numeru zlecenia
           "DB_Data".Stanowisko1.Production.OrderNo := 0;
           "DB_Data".Stanowisko1.Production.ProductNo := 0;

           //Zerowanie flagi ladowania
           "DB_Data".Stanowisko1.Stats.Loaded := 0;

           //Sprawdzenie czy jest zlecenie (numer int = 0 -> brak zlecenia)
           IF "DB_Zlecenia".NastepneZlecenie.Zlecenie.ID = 0 THEN
               //Brak zlecenia - Start zablokowany
               "DB_Data".Stanowisko1.Commands.Start.Enable := 0;
               "DB_Data".Stanowisko1.Stats.Instruction := 0;
           ELSE
               //Jest zlecenie
               "DB_Data".Stanowisko1.Stats.Instruction := 1;

               //Przejscie do montazu jezeli paletka jest aktywna i start klikniety
               IF "DB_Data".Stanowisko1.Sensors.PalletPresent THEN
                   "DB_Data".Stanowisko1.Commands.Start.Enable := 1;
                   IF "DB_Data".Stanowisko1.Commands.Start.State THEN
                       "DB_Data".Stanowisko1.Production.State := 1;
                       "DB_Data".Stanowisko1.Commands.Start.State := 0;
                       "DB_Data".Stanowisko1.MontazState := 0;
                   END_IF;
               ELSE
                   "DB_Data".Stanowisko1.Commands.Start.Enable := 0;
               END_IF;
           END_IF;

       1:
           //Ustawienie przycisków
           "DB_Data".Stanowisko1.Commands.Start.Enable := 0;
           "DB_Data".Stanowisko1.Commands.AbortProcess.Enable := 1;
           "DB_Data".Stanowisko1.Commands.FInish.Enable := 1;
           "DB_Data".Stanowisko1.Commands.ReportFault.Enable := 1;

           CASE "DB_Data".Stanowisko1.MontazState OF
                   //Ustawienie wartosci przed montazem
               0:
                   "DB_Data".Stanowisko1.Production.OrderNo := "DB_Zlecenia".NastepneZlecenie.Zlecenie.ID;
                   "DB_Data".Stanowisko1.Production.ProductNo := "DB_Zlecenia".NastepneZlecenie.Zlecenie.PartNo;
                   "DB_Data".Stanowisko1.Stats.Instruction := "DB_Zlecenia".NastepneZlecenie.Zlecenie.Model; //Modele od 2 do 8 (0-1 zarezerwowane dla informacji)
                   #temp_start_time := RD_LOC_T(OUT => "DB_Zlecenia".NastepneZlecenie.Zlecenie."Time".Stanowisko1.StartTime); // Zapis czasu rozpoczecia

                   CASE "DB_Zlecenia".NastepneZlecenie.Zlecenie.Model OF
                       2:
                           "DB_Zlecenia".NastepneZlecenie.Zlecenie."Time".Stanowisko1.TargetTime := 54;
                           "DB_Zlecenia".NastepneZlecenie.Zlecenie."Time".Stanowisko2.TargetTime := 60;
                           "DB_Zlecenia".NastepneZlecenie.Zlecenie."Time".Stanowisko3.TargetTime := 52;
                           "DB_Zlecenia".NastepneZlecenie.Zlecenie."Time".StanowiskoQC.TargetTime := 15;
                       3:
                           "DB_Zlecenia".NastepneZlecenie.Zlecenie."Time".Stanowisko1.TargetTime := 39;
                           "DB_Zlecenia".NastepneZlecenie.Zlecenie."Time".Stanowisko2.TargetTime := 42;
                           "DB_Zlecenia".NastepneZlecenie.Zlecenie."Time".Stanowisko3.TargetTime := 66;
                           "DB_Zlecenia".NastepneZlecenie.Zlecenie."Time".StanowiskoQC.TargetTime := 15;
                       4:
                           "DB_Zlecenia".NastepneZlecenie.Zlecenie."Time".Stanowisko1.TargetTime := 26;
                           "DB_Zlecenia".NastepneZlecenie.Zlecenie."Time".Stanowisko2.TargetTime := 82;
                           "DB_Zlecenia".NastepneZlecenie.Zlecenie."Time".Stanowisko3.TargetTime := 59;
                           "DB_Zlecenia".NastepneZlecenie.Zlecenie."Time".StanowiskoQC.TargetTime := 15;
                       5:
                           "DB_Zlecenia".NastepneZlecenie.Zlecenie."Time".Stanowisko1.TargetTime := 27;
                           "DB_Zlecenia".NastepneZlecenie.Zlecenie."Time".Stanowisko2.TargetTime := 29;
                           "DB_Zlecenia".NastepneZlecenie.Zlecenie."Time".Stanowisko3.TargetTime := 53;
                           "DB_Zlecenia".NastepneZlecenie.Zlecenie."Time".StanowiskoQC.TargetTime := 15;
                       6:
                           "DB_Zlecenia".NastepneZlecenie.Zlecenie."Time".Stanowisko1.TargetTime := 30;
                           "DB_Zlecenia".NastepneZlecenie.Zlecenie."Time".Stanowisko2.TargetTime := 33;
                           "DB_Zlecenia".NastepneZlecenie.Zlecenie."Time".Stanowisko3.TargetTime := 55;
                           "DB_Zlecenia".NastepneZlecenie.Zlecenie."Time".StanowiskoQC.TargetTime := 15;
                       7:
                           "DB_Zlecenia".NastepneZlecenie.Zlecenie."Time".Stanowisko1.TargetTime := 20;
                           "DB_Zlecenia".NastepneZlecenie.Zlecenie."Time".Stanowisko2.TargetTime := 33;
                           "DB_Zlecenia".NastepneZlecenie.Zlecenie."Time".Stanowisko3.TargetTime := 43;
                           "DB_Zlecenia".NastepneZlecenie.Zlecenie."Time".StanowiskoQC.TargetTime := 15;
                   END_CASE;

                   //"RFID_test".Bufor_Zapis
                   "RFID_test".Bufor_Zapis[0] := INT_TO_BYTE("DB_Zlecenia".NastepneZlecenie.Zlecenie.ID);
                   "RFID_test".Bufor_Zapis[1] := INT_TO_BYTE("DB_Zlecenia".NastepneZlecenie.Zlecenie.Model);
                   "RFID_test".Bufor_Zapis[2] := INT_TO_BYTE("DB_Zlecenia".NastepneZlecenie.Zlecenie.PartNo);
                   "DB_Data".Stanowisko1.Sensors.RFID.CmdWrite := TRUE;

                   "DB_Data".Stanowisko1.MontazState := 1;

               1:
                   #temp_taget_time := "DB_Zlecenia".NastepneZlecenie.Zlecenie."Time".Stanowisko1.TargetTime;

                   "DB_Data".Stanowisko1.Sensors.RFID.CmdWrite := FALSE;

                   "DB_Data".Stanowisko1."Time".RemainingSec := "DB_Zlecenia".NastepneZlecenie.Zlecenie."Time".Stanowisko1.TargetTime;
                   "DB_Data".Stanowisko1."Time".Blink := FALSE;

                   "DB_Data".Stanowisko1.MontazState := 2;

               2:
                   #Status_Czasu := RD_SYS_T(OUT => #Czas_DTL);

                   IF #Czas_DTL.SECOND <> "DB_Data".Stanowisko1."Time".LastSec THEN
                       "DB_Data".Stanowisko1."Time".LastSec := #Czas_DTL.SECOND;

                       IF "DB_Data".Stanowisko1."Time".RemainingSec > 0 THEN
                           "DB_Data".Stanowisko1."Time".RemainingSec := "DB_Data".Stanowisko1."Time".RemainingSec - 1;
                       END_IF;

                       IF "DB_Data".Stanowisko1."Time".RemainingSec <= 0 THEN
                           "DB_Data".Stanowisko1."Time".Blink := NOT "DB_Data".Stanowisko1."Time".Blink;
                       END_IF;
                   END_IF;

                   #Minuty := "DB_Data".Stanowisko1."Time".RemainingSec / 60;
                   #Sekundy := "DB_Data".Stanowisko1."Time".RemainingSec MOD 60;

                   #StrMin := INT_TO_STRING(#Minuty);
                   #StrSec := INT_TO_STRING(#Sekundy);

                   #StrMin := RIGHT(IN := #StrMin, L := LEN(#StrMin) - 1);
                   #StrSec := RIGHT(IN := #StrSec, L := LEN(#StrSec) - 1);

